gfCNCPoint5[18041] = {X 248.0563, Y 60.9282, Z -7.1667, A 0.000, B 0.000, C 0.000 }
gfCNCPoint5[18042] = {X 275.7918, Y 71.9370, Z -7.1667, A 0.000, B 0.000, C 0.000 }
gfCNCPoint5[18043] = {X 275.7935, Y 63.0708, Z -7.1667, A 0.000, B 0.000, C 0.000 }
gfCNCPoint5[18044] = {X 275.6909, Y 63.0586, Z -7.1667, A 0.000, B 0.000, C 0.000 }
gfCNCPoint5[18045] = {X 275.5887, Y 63.0439, Z -7.1667, A 0.000, B 0.000, C 0.000 }
gfCNCPoint5[18046] = {X 274.6513, Y 62.7818, Z -7.1667, A 0.000, B 0.000, C 0.000 }
gfCNCPoint5[18047] = {X 273.8005, Y 62.3090, Z -7.1667, A 0.000, B 0.000, C 0.000 }
gfCNCPoint5[18048] = {X 273.0828, Y 61.6514, Z -7.1667, A 0.000, B 0.000, C 0.000 }
gfCNCPoint5[18049] = {X 272.5376, Y 60.8451, Z -7.1667, A 0.000, B 0.000, C 0.000 }
gfCNCPoint5[18050] = {X 272.1947, Y 59.9341, Z -7.1667, A 0.000, B 0.000, C 0.000 }
gfCNCPoint5[18051] = {X 272.0728, Y 58.9684, Z -7.1667, A 0.000, B 0.000, C 0.000 }
gfCNCPoint5[18052] = {X 272.0727, Y 58.0000, Z -7.1667, A 0.000, B 0.000, C 0.000 }
gfCNCPoint5[18053] = {X 272.1770, Y 57.0743, Z -7.1667, A 0.000, B 0.000, C 0.000 }
gfCNCPoint5[18054] = {X 272.4847, Y 56.1950, Z -7.1667, A 0.000, B 0.000, C 0.000 }
gfCNCPoint5[18055] = {X 272.9803, Y 55.4063, Z -7.1667, A 0.000, B 0.000, C 0.000 }
gfCNCPoint5[18056] = {X 273.6390, Y 54.7476, Z -7.1667, A 0.000, B 0.000, C 0.000 }
gfCNCPoint5[18057] = {X 274.4277, Y 54.2520, Z -7.1667, A 0.000, B 0.000, C 0.000 }
gfCNCPoint5[18058] = {X 275.3070, Y 53.9443, Z -7.1667, A 0.000, B 0.000, C 0.000 }
gfCNCPoint5[18059] = {X 276.2327, Y 53.8400, Z -7.1667, A 0.000, B 0.000, C 0.000 }
gfCNCPoint5[18060] = {X 292.7731, Y 53.8400, Z -7.1667, A 0.000, B 0.000, C 0.000 }
gfCNCPoint5[18061] = {X 293.6988, Y 53.9443, Z -7.1667, A 0.000, B 0.000, C 0.000 }
gfCNCPoint5[18062] = {X 294.5780, Y 54.2520, Z -7.1667, A 0.000, B 0.000, C 0.000 }
gfCNCPoint5[18063] = {X 295.3668, Y 54.7476, Z -7.1667, A 0.000, B 0.000, C 0.000 }
gfCNCPoint5[18064] = {X 296.0255, Y 55.4063, Z -7.1667, A 0.000, B 0.000, C 0.000 }
gfCNCPoint5[18065] = {X 296.5211, Y 56.1950, Z -7.1667, A 0.000, B 0.000, C 0.000 }
gfCNCPoint5[18066] = {X 296.8288, Y 57.0743, Z -7.1667, A 0.000, B 0.000, C 0.000 }
gfCNCPoint5[18067] = {X 296.9331, Y 58.0000, Z -7.1667, A 0.000, B 0.000, C 0.000 }
gfCNCPoint5[18068] = {X 296.9331, Y 58.9345, Z -7.1667, A 0.000, B 0.000, C 0.000 }
gfCNCPoint5[18069] = {X 296.8157, Y 59.9063, Z -7.1667, A 0.000, B 0.000, C 0.000 }
gfCNCPoint5[18070] = {X 296.4753, Y 60.8241, Z -7.1667, A 0.000, B 0.000, C 0.000 }
gfCNCPoint5[18071] = {X 295.9306, Y 61.6374, Z -7.1667, A 0.000, B 0.000, C 0.000 }
gfCNCPoint5[18072] = {X 295.2116, Y 62.3015, Z -7.1667, A 0.000, B 0.000, C 0.000 }
gfCNCPoint5[18073] = {X 294.3577, Y 62.7801, Z -7.1667, A 0.000, B 0.000, C 0.000 }
gfCNCPoint5[18074] = {X 293.4159, Y 63.0468, Z -7.1667, A 0.000, B 0.000, C 0.000 }
gfCNCPoint5[18075] = {X 293.3191, Y 63.0611, Z -7.1667, A 0.000, B 0.000, C 0.000 }
gfCNCPoint5[18076] = {X 293.2221, Y 63.0731, Z -7.1667, A 0.000, B 0.000, C 0.000 }
gfCNCPoint5[18077] = {X 293.2138, Y 63.1615, Z -7.1667, A 0.000, B 0.000, C 0.000 }
gfCNCPoint5[18078] = {X 293.2249, Y 92.9203, Z -7.1667, A 0.000, B 0.000, C 0.000 }
gfCNCPoint5[18079] = {X 293.3202, Y 92.9325, Z -7.1667, A 0.000, B 0.000, C 0.000 }
gfCNCPoint5[18080] = {X 293.4152, Y 92.9468, Z -7.1667, A 0.000, B 0.000, C 0.000 }
gfCNCPoint5[18081] = {X 294.3566, Y 93.2161, Z -7.1667, A 0.000, B 0.000, C 0.000 }
gfCNCPoint5[18082] = {X 295.2099, Y 93.6965, Z -7.1667, A 0.000, B 0.000, C 0.000 }
gfCNCPoint5[18083] = {X 295.9285, Y 94.3617, Z -7.1667, A 0.000, B 0.000, C 0.000 }
gfCNCPoint5[18084] = {X 296.4732, Y 95.1754, Z -7.1667, A 0.000, B 0.000, C 0.000 }
gfCNCPoint5[18085] = {X 296.8142, Y 96.0933, Z -7.1667, A 0.000, B 0.000, C 0.000 }
gfCNCPoint5[18086] = {X 296.9331, Y 97.0653, Z -7.1667, A 0.000, B 0.000, C 0.000 }
gfCNCPoint5[18087] = {X 296.9331, Y 98.0000, Z -7.1667, A 0.000, B 0.000, C 0.000 }
gfCNCPoint5[18088] = {X 296.8288, Y 98.9257, Z -7.1667, A 0.000, B 0.000, C 0.000 }
gfCNCPoint5[18089] = {X 296.5211, Y 99.8050, Z -7.1667, A 0.000, B 0.000, C 0.000 }
gfCNCPoint5[18090] = {X 296.0255, Y 100.5937, Z -7.1667, A 0.000, B 0.000, C 0.000 }
gfCNCPoint5[18091] = {X 295.3668, Y 101.2524, Z -7.1667, A 0.000, B 0.000, C 0.000 }
gfCNCPoint5[18092] = {X 294.5780, Y 101.7480, Z -7.1667, A 0.000, B 0.000, C 0.000 }
gfCNCPoint5[18093] = {X 293.6988, Y 102.0557, Z -7.1667, A 0.000, B 0.000, C 0.000 }
gfCNCPoint5[18094] = {X 292.7731, Y 102.1600, Z -7.1667, A 0.000, B 0.000, C 0.000 }
gfCNCPoint5[18095] = {X 276.2327, Y 102.1600, Z -7.1667, A 0.000, B 0.000, C 0.000 }
gfCNCPoint5[18096] = {X 275.3070, Y 102.0557, Z -7.1667, A 0.000, B 0.000, C 0.000 }
gfCNCPoint5[18097] = {X 274.4277, Y 101.7480, Z -7.1667, A 0.000, B 0.000, C 0.000 }
gfCNCPoint5[18098] = {X 273.6390, Y 101.2524, Z -7.1667, A 0.000, B 0.000, C 0.000 }
gfCNCPoint5[18099] = {X 272.9803, Y 100.5937, Z -7.1667, A 0.000, B 0.000, C 0.000 }
gfCNCPoint5[18100] = {X 272.4847, Y 99.8050, Z -7.1667, A 0.000, B 0.000, C 0.000 }
gfCNCPoint5[18101] = {X 272.1770, Y 98.9257, Z -7.1667, A 0.000, B 0.000, C 0.000 }
gfCNCPoint5[18102] = {X 272.0727, Y 98.0000, Z -7.1667, A 0.000, B 0.000, C 0.000 }
gfCNCPoint5[18103] = {X 272.0727, Y 97.0658, Z -7.1667, A 0.000, B 0.000, C 0.000 }
gfCNCPoint5[18104] = {X 272.1634, Y 96.2021, Z -7.1667, A 0.000, B 0.000, C 0.000 }
gfCNCPoint5[18105] = {X 272.4314, Y 95.3761, Z -7.1667, A 0.000, B 0.000, C 0.000 }
gfCNCPoint5[18106] = {X 272.8651, Y 94.6237, Z -7.1667, A 0.000, B 0.000, C 0.000 }
gfCNCPoint5[18107] = {X 273.4455, Y 93.9777, Z -7.1667, A 0.000, B 0.000, C 0.000 }
gfCNCPoint5[18108] = {X 274.1475, Y 93.4663, Z -7.1667, A 0.000, B 0.000, C 0.000 }
gfCNCPoint5[18109] = {X 274.9403, Y 93.1118, Z -7.1667, A 0.000, B 0.000, C 0.000 }
gfCNCPoint5[18110] = {X 275.7894, Y 92.9296, Z -7.1667, A 0.000, B 0.000, C 0.000 }
gfCNCPoint5[18111] = {X 275.7894, Y 85.4858, Z -7.1667, A 0.000, B 0.000, C 0.000 }
gfCNCPoint5[18112] = {X 262.6229, Y 80.3245, Z -7.1667, A 0.000, B 0.000, C 0.000 }
gfCNCPoint5[18113] = {X 262.1919, Y 80.5968, Z -7.1667, A 0.000, B 0.000, C 0.000 }
gfCNCPoint5[18114] = {X 237.6370, Y 96.5016, Z -7.1667, A 0.000, B 0.000, C 0.000 }
gfCNCPoint5[18115] = {X 237.6398, Y 97.0655, Z -7.1667, A 0.000, B 0.000, C 0.000 }
gfCNCPoint5[18116] = {X 237.6398, Y 98.0000, Z -7.1667, A 0.000, B 0.000, C 0.000 }
gfCNCPoint5[18117] = {X 237.5355, Y 98.9257, Z -7.1667, A 0.000, B 0.000, C 0.000 }
gfCNCPoint5[18118] = {X 237.2278, Y 99.8050, Z -7.1667, A 0.000, B 0.000, C 0.000 }
gfCNCPoint5[18119] = {X 236.7322, Y 100.5937, Z -7.1667, A 0.000, B 0.000, C 0.000 }
gfCNCPoint5[18120] = {X 236.0735, Y 101.2524, Z -7.1667, A 0.000, B 0.000, C 0.000 }
gfCNCPoint5[18121] = {X 235.2847, Y 101.7480, Z -7.1667, A 0.000, B 0.000, C 0.000 }
gfCNCPoint5[18122] = {X 234.4055, Y 102.0557, Z -7.1667, A 0.000, B 0.000, C 0.000 }
gfCNCPoint5[18123] = {X 233.4798, Y 102.1600, Z -7.1667, A 0.000, B 0.000, C 0.000 }
gfCNCPoint5[18124] = {X 214.1790, Y 102.1600, Z -7.1667, A 0.000, B 0.000, C 0.000 }
gfCNCPoint5[18125] = {X 213.7860, Y 102.1414, Z -7.1667, A 0.000, B 0.000, C 0.000 }
gfCNCPoint5[18126] = {X 213.3966, Y 102.0857, Z -7.1667, A 0.000, B 0.000, C 0.000 }
gfCNCPoint5[18127] = {X 213.0071, Y 102.1414, Z -7.1667, A 0.000, B 0.000, C 0.000 }
gfCNCPoint5[18128] = {X 212.6141, Y 102.1600, Z -7.1667, A 0.000, B 0.000, C 0.000 }
gfCNCPoint5[18129] = {X 194.9870, Y 102.1600, Z -7.1667, A 0.000, B 0.000, C 0.000 }
gfCNCPoint5[18130] = {X 194.0613, Y 102.0557, Z -7.1667, A 0.000, B 0.000, C 0.000 }
gfCNCPoint5[18131] = {X 193.1820, Y 101.7480, Z -7.1667, A 0.000, B 0.000, C 0.000 }
gfCNCPoint5[18132] = {X 192.3932, Y 101.2524, Z -7.1667, A 0.000, B 0.000, C 0.000 }
gfCNCPoint5[18133] = {X 191.7345, Y 100.5937, Z -7.1667, A 0.000, B 0.000, C 0.000 }
gfCNCPoint5[18134] = {X 191.2389, Y 99.8050, Z -7.1667, A 0.000, B 0.000, C 0.000 }
gfCNCPoint5[18135] = {X 190.9313, Y 98.9257, Z -7.1667, A 0.000, B 0.000, C 0.000 }
gfCNCPoint5[18136] = {X 190.8270, Y 98.0000, Z -7.1667, A 0.000, B 0.000, C 0.000 }
gfCNCPoint5[18137] = {X 190.8270, Y 97.0659, Z -7.1667, A 0.000, B 0.000, C 0.000 }
gfCNCPoint5[18138] = {X 190.9241, Y 96.1723, Z -7.1667, A 0.000, B 0.000, C 0.000 }
gfCNCPoint5[18139] = {X 191.2109, Y 95.3203, Z -7.1667, A 0.000, B 0.000, C 0.000 }
gfCNCPoint5[18140] = {X 191.6741, Y 94.5499, Z -7.1667, A 0.000, B 0.000, C 0.000 }
gfCNCPoint5[18141] = {X 191.7354, Y 94.4712, Z -7.1667, A 0.000, B 0.000, C 0.000 }
gfCNCPoint5[18142] = {X 191.7986, Y 94.3939, Z -7.1667, A 0.000, B 0.000, C 0.000 }
gfCNCPoint5[18143] = {X 188.6351, Y 90.9402, Z -7.1667, A 0.000, B 0.000, C 0.000 }
gfCNCPoint5[18144] = {X 150.0187, Y 90.9402, Z -7.1667, A 0.000, B 0.000, C 0.000 }
gfCNCPoint5[18145] = {X 146.9341, Y 94.3576, Z -7.1667, A 0.000, B 0.000, C 0.000 }
gfCNCPoint5[18146] = {X 147.4805, Y 95.1722, Z -7.1667, A 0.000, B 0.000, C 0.000 }
gfCNCPoint5[18147] = {X 147.8218, Y 96.0918, Z -7.1667, A 0.000, B 0.000, C 0.000 }
gfCNCPoint5[18148] = {X 147.9391, Y 97.0657, Z -7.1667, A 0.000, B 0.000, C 0.000 }
gfCNCPoint5[18149] = {X 147.9391, Y 98.0000, Z -7.1667, A 0.000, B 0.000, C 0.000 }
gfCNCPoint5[18150] = {X 147.8348, Y 98.9257, Z -7.1667, A 0.000, B 0.000, C 0.000 }
gfCNCPoint5[18151] = {X 147.5271, Y 99.8050, Z -7.1667, A 0.000, B 0.000, C 0.000 }
gfCNCPoint5[18152] = {X 147.0315, Y 100.5937, Z -7.1667, A 0.000, B 0.000, C 0.000 }
gfCNCPoint5[18153] = {X 146.3728, Y 101.2524, Z -7.1667, A 0.000, B 0.000, C 0.000 }
gfCNCPoint5[18154] = {X 145.5841, Y 101.7480, Z -7.1667, A 0.000, B 0.000, C 0.000 }
gfCNCPoint5[18155] = {X 144.7048, Y 102.0557, Z -7.1667, A 0.000, B 0.000, C 0.000 }
gfCNCPoint5[18156] = {X 143.7791, Y 102.1600, Z -7.1667, A 0.000, B 0.000, C 0.000 }
gfCNCPoint5[18157] = {X 125.0000, Y 102.1600, Z -7.1667, A 0.000, B 0.000, C 0.000 }
gfCNCPoint5[18158] = {X 124.0743, Y 102.0557, Z -7.1667, A 0.000, B 0.000, C 0.000 }
gfCNCPoint5[18159] = {X 123.1950, Y 101.7480, Z -7.1667, A 0.000, B 0.000, C 0.000 }
gfCNCPoint5[18160] = {X 122.4063, Y 101.2524, Z -7.1667, A 0.000, B 0.000, C 0.000 }
gfCNCPoint5[18161] = {X 121.7476, Y 100.5937, Z -7.1667, A 0.000, B 0.000, C 0.000 }
gfCNCPoint5[18162] = {X 121.2520, Y 99.8050, Z -7.1667, A 0.000, B 0.000, C 0.000 }
gfCNCPoint5[18163] = {X 120.9443, Y 98.9257, Z -7.1667, A 0.000, B 0.000, C 0.000 }
gfCNCPoint5[18164] = {X 120.8400, Y 98.0000, Z -7.1667, A 0.000, B 0.000, C 0.000 }
gfCNCPoint5[18165] = {X 120.8400, Y 97.0659, Z -7.1667, A 0.000, B 0.000, C 0.000 }
gfCNCPoint5[18166] = {X 120.9405, Y 96.1569, Z -7.1667, A 0.000, B 0.000, C 0.000 }
gfCNCPoint5[18167] = {X 121.2373, Y 95.2918, Z -7.1667, A 0.000, B 0.000, C 0.000 }
gfCNCPoint5[18168] = {X 121.7159, Y 94.5125, Z -7.1667, A 0.000, B 0.000, C 0.000 }
gfCNCPoint5[18169] = {X 122.3532, Y 93.8566, Z -7.1667, A 0.000, B 0.000, C 0.000 }
gfCNCPoint5[18170] = {X 123.1185, Y 93.3558, Z -7.1667, A 0.000, B 0.000, C 0.000 }
gfCNCPoint5[18171] = {X 123.9747, Y 93.0343, Z -7.1667, A 0.000, B 0.000, C 0.000 }
gfCNCPoint5[18172] = {X 124.8804, Y 92.9077, Z -7.1667, A 0.000, B 0.000, C 0.000 }
gfCNCPoint5[18173] = {X 124.9141, Y 92.8889, Z -7.1667, A 0.000, B 0.000, C 0.000 }
gfCNCPoint5[18174] = {X 124.9512, Y 92.8787, Z -7.1667, A 0.000, B 0.000, C 0.000 }
gfCNCPoint5[18175] = {X 125.4723, Y 92.8015, Z -7.1667, A 0.000, B 0.000, C 0.000 }
gfCNCPoint5[18176] = {X 126.3315, Y 92.6561, Z -7.1667, A 0.000, B 0.000, C 0.000 }
gfCNCPoint5[18177] = {X 127.1785, Y 92.4511, Z -7.1667, A 0.000, B 0.000, C 0.000 }
gfCNCPoint5[18178] = {X 128.3866, Y 91.3174, Z -7.1667, A 0.000, B 0.000, C 0.000 }
gfCNCPoint5[18179] = {X 129.5302, Y 90.1187, Z -7.1667, A 0.000, B 0.000, C 0.000 }
gfCNCPoint5[18180] = {X 140.7977, Y 77.7462, Z -7.1667, A 0.000, B 0.000, C 0.000 }
gfCNCPoint5[18181] = {X 137.8403, Y 75.0529, Z -7.1667, A 0.000, B 0.000, C 0.000 }
gfCNCPoint5[18182] = {X 140.8568, Y 77.8000, Z -7.1667, A 0.000, B 0.000, C 0.000 }
gfCNCPoint5[18183] = {X 155.9346, Y 61.2436, Z -7.1667, A 0.000, B 0.000, C 0.000 }
gfCNCPoint5[18184] = {X 155.5463, Y 60.5376, Z -7.1667, A 0.000, B 0.000, C 0.000 }
gfCNCPoint5[18185] = {X 155.3043, Y 59.7689, Z -7.1667, A 0.000, B 0.000, C 0.000 }
gfCNCPoint5[18186] = {X 155.2181, Y 58.9678, Z -7.1667, A 0.000, B 0.000, C 0.000 }
gfCNCPoint5[18187] = {X 155.2180, Y 58.0000, Z -7.1667, A 0.000, B 0.000, C 0.000 }
gfCNCPoint5[18188] = {X 155.3203, Y 57.0921, Z -7.1667, A 0.000, B 0.000, C 0.000 }
gfCNCPoint5[18189] = {X 155.6220, Y 56.2298, Z -7.1667, A 0.000, B 0.000, C 0.000 }
gfCNCPoint5[18190] = {X 156.1081, Y 55.4562, Z -7.1667, A 0.000, B 0.000, C 0.000 }
gfCNCPoint5[18191] = {X 156.7541, Y 54.8101, Z -7.1667, A 0.000, B 0.000, C 0.000 }
gfCNCPoint5[18192] = {X 157.5277, Y 54.3240, Z -7.1667, A 0.000, B 0.000, C 0.000 }
gfCNCPoint5[18193] = {X 158.3901, Y 54.0223, Z -7.1667, A 0.000, B 0.000, C 0.000 }
gfCNCPoint5[18194] = {X 159.2980, Y 53.9200, Z -7.1667, A 0.000, B 0.000, C 0.000 }
gfCNCPoint5[18195] = {X 178.5335, Y 53.9200, Z -7.1667, A 0.000, B 0.000, C 0.000 }
gfCNCPoint5[18196] = {X 179.4414, Y 54.0223, Z -7.1667, A 0.000, B 0.000, C 0.000 }
gfCNCPoint5[18197] = {X 180.3037, Y 54.3240, Z -7.1667, A 0.000, B 0.000, C 0.000 }
gfCNCPoint5[18198] = {X 181.0773, Y 54.8101, Z -7.1667, A 0.000, B 0.000, C 0.000 }
gfCNCPoint5[18199] = {X 181.7234, Y 55.4562, Z -7.1667, A 0.000, B 0.000, C 0.000 }
gfCNCPoint5[18200] = {X 182.2095, Y 56.2298, Z -7.1667, A 0.000, B 0.000, C 0.000 }
gfCNCPoint5[18201] = {X 182.5112, Y 57.0921, Z -7.1667, A 0.000, B 0.000, C 0.000 }
gfCNCPoint5[18202] = {X 182.6135, Y 58.0000, Z -7.1667, A 0.000, B 0.000, C 0.000 }
gfCNCPoint5[18203] = {X 182.6135, Y 58.9342, Z -7.1667, A 0.000, B 0.000, C 0.000 }
gfCNCPoint5[18204] = {X 182.5335, Y 59.7381, Z -7.1667, A 0.000, B 0.000, C 0.000 }
gfCNCPoint5[18205] = {X 182.2967, Y 60.5104, Z -7.1667, A 0.000, B 0.000, C 0.000 }
gfCNCPoint5[18206] = {X 181.9123, Y 61.2210, Z -7.1667, A 0.000, B 0.000, C 0.000 }
gfCNCPoint5[18207] = {X 209.1194, Y 90.9217, Z -7.1667, A 0.000, B 0.000, C 0.000 }
gfCNCPoint5[18208] = {X 209.7993, Y 91.6258, Z -7.1667, A 0.000, B 0.000, C 0.000 }
gfCNCPoint5[18209] = {X 210.5151, Y 92.2933, Z -7.1667, A 0.000, B 0.000, C 0.000 }
gfCNCPoint5[18210] = {X 210.9595, Y 92.5941, Z -7.1667, A 0.000, B 0.000, C 0.000 }
gfCNCPoint5[18211] = {X 211.4659, Y 92.7713, Z -7.1667, A 0.000, B 0.000, C 0.000 }
gfCNCPoint5[18212] = {X 212.0678, Y 92.8979, Z -7.1667, A 0.000, B 0.000, C 0.000 }
gfCNCPoint5[18213] = {X 213.3902, Y 93.0645, Z -7.1667, A 0.000, B 0.000, C 0.000 }
gfCNCPoint5[18214] = {X 213.4129, Y 93.0582, Z -7.1667, A 0.000, B 0.000, C 0.000 }
gfCNCPoint5[18215] = {X 214.4629, Y 92.9753, Z -7.1667, A 0.000, B 0.000, C 0.000 }
gfCNCPoint5[18216] = {X 215.5144, Y 92.9145, Z -7.1667, A 0.000, B 0.000, C 0.000 }
gfCNCPoint5[18217] = {X 216.2276, Y 92.8363, Z -7.1667, A 0.000, B 0.000, C 0.000 }
gfCNCPoint5[18218] = {X 216.9142, Y 92.6283, Z -7.1667, A 0.000, B 0.000, C 0.000 }
gfCNCPoint5[18219] = {X 217.5510, Y 92.2978, Z -7.1667, A 0.000, B 0.000, C 0.000 }
gfCNCPoint5[18220] = {X 223.0910, Y 88.7225, Z -7.1667, A 0.000, B 0.000, C 0.000 }
gfCNCPoint5[18221] = {X 246.3530, Y 73.8482, Z -7.1667, A 0.000, B 0.000, C 0.000 }
gfCNCPoint5[18222] = {X 221.7196, Y 64.1819, Z -7.1667, A 0.000, B 0.000, C 0.000 }
gfCNCPoint5[18223] = {X 219.9261, Y 63.5817, Z -7.1667, A 0.000, B 0.000, C 0.000 }
gfCNCPoint5[18224] = {X 218.0758, Y 63.1899, Z -7.1667, A 0.000, B 0.000, C 0.000 }
gfCNCPoint5[18225] = {X 216.1929, Y 63.0117, Z -7.1667, A 0.000, B 0.000, C 0.000 }
gfCNCPoint5[18226] = {X 215.3127, Y 62.8850, Z -7.1667, A 0.000, B 0.000, C 0.000 }
gfCNCPoint5[18227] = {X 214.4809, Y 62.5706, Z -7.1667, A 0.000, B 0.000, C 0.000 }
gfCNCPoint5[18228] = {X 213.7369, Y 62.0834, Z -7.1667, A 0.000, B 0.000, C 0.000 }
gfCNCPoint5[18229] = {X 213.1162, Y 61.4466, Z -7.1667, A 0.000, B 0.000, C 0.000 }
gfCNCPoint5[18230] = {X 212.6482, Y 60.6905, Z -7.1667, A 0.000, B 0.000, C 0.000 }
gfCNCPoint5[18231] = {X 212.3552, Y 59.8509, Z -7.1667, A 0.000, B 0.000, C 0.000 }
gfCNCPoint5[18232] = {X 212.2509, Y 58.9678, Z -7.1667, A 0.000, B 0.000, C 0.000 }
gfCNCPoint5[18233] = {X 212.2508, Y 58.0000, Z -7.1667, A 0.000, B 0.000, C 0.000 }
gfCNCPoint5[18234] = {X 212.3531, Y 57.0921, Z -7.1667, A 0.000, B 0.000, C 0.000 }
gfCNCPoint5[18235] = {X 212.6549, Y 56.2298, Z -7.1667, A 0.000, B 0.000, C 0.000 }
gfCNCPoint5[18236] = {X 213.1409, Y 55.4562, Z -7.1667, A 0.000, B 0.000, C 0.000 }
gfCNCPoint5[18237] = {X 213.7870, Y 54.8101, Z -7.1667, A 0.000, B 0.000, C 0.000 }
gfCNCPoint5[18238] = {X 214.5606, Y 54.3240, Z -7.1667, A 0.000, B 0.000, C 0.000 }
gfCNCPoint5[18239] = {X 215.4229, Y 54.0223, Z -7.1667, A 0.000, B 0.000, C 0.000 }
gfCNCPoint5[18240] = {X 216.3308, Y 53.9200, Z -7.1667, A 0.000, B 0.000, C 0.000 }
gfCNCPoint5[18241] = {X 237.2617, Y 53.9200, Z -7.1667, A 0.000, B 0.000, C 0.000 }
gfCNCPoint5[18242] = {X 238.1696, Y 54.0223, Z -7.1667, A 0.000, B 0.000, C 0.000 }
gfCNCPoint5[18243] = {X 239.0319, Y 54.3240, Z -7.1667, A 0.000, B 0.000, C 0.000 }
gfCNCPoint5[18244] = {X 239.8055, Y 54.8101, Z -7.1667, A 0.000, B 0.000, C 0.000 }
gfCNCPoint5[18245] = {X 240.4516, Y 55.4562, Z -7.1667, A 0.000, B 0.000, C 0.000 }
gfCNCPoint5[18246] = {X 240.9376, Y 56.2298, Z -7.1667, A 0.000, B 0.000, C 0.000 }
gfCNCPoint5[18247] = {X 241.2394, Y 57.0921, Z -7.1667, A 0.000, B 0.000, C 0.000 }
gfCNCPoint5[18248] = {X 241.3417, Y 58.0000, Z -7.1667, A 0.000, B 0.000, C 0.000 }
gfCNCPoint5[18249] = {X 241.3417, Y 58.3958, Z -7.1667, A 0.000, B 0.000, C 0.000 }
gfCNCPoint5[18250] = {X 248.0270, Y 61.0026, Z -7.1667, A 0.000, B 0.000, C 0.000 }
gfCNCPoint5[18251] = {X 275.8718, Y 72.0548, Z -7.1667, A 0.000, B 0.000, C 0.000 }
gfCNCPoint5[18252] = {X 275.8735, Y 62.9982, Z -7.1667, A 0.000, B 0.000, C 0.000 }
gfCNCPoint5[18253] = {X 275.7370, Y 62.9838, Z -7.1667, A 0.000, B 0.000, C 0.000 }
gfCNCPoint5[18254] = {X 275.6011, Y 62.9649, Z -7.1667, A 0.000, B 0.000, C 0.000 }
gfCNCPoint5[18255] = {X 274.6817, Y 62.7078, Z -7.1667, A 0.000, B 0.000, C 0.000 }
gfCNCPoint5[18256] = {X 273.8473, Y 62.2441, Z -7.1667, A 0.000, B 0.000, C 0.000 }
gfCNCPoint5[18257] = {X 273.1434, Y 61.5992, Z -7.1667, A 0.000, B 0.000, C 0.000 }
gfCNCPoint5[18258] = {X 272.6087, Y 60.8083, Z -7.1667, A 0.000, B 0.000, C 0.000 }
gfCNCPoint5[18259] = {X 272.2723, Y 59.9149, Z -7.1667, A 0.000, B 0.000, C 0.000 }
gfCNCPoint5[18260] = {X 272.1528, Y 58.9678, Z -7.1667, A 0.000, B 0.000, C 0.000 }
gfCNCPoint5[18261] = {X 272.1527, Y 58.0000, Z -7.1667, A 0.000, B 0.000, C 0.000 }
gfCNCPoint5[18262] = {X 272.2550, Y 57.0921, Z -7.1667, A 0.000, B 0.000, C 0.000 }
gfCNCPoint5[18263] = {X 272.5567, Y 56.2298, Z -7.1667, A 0.000, B 0.000, C 0.000 }
gfCNCPoint5[18264] = {X 273.0428, Y 55.4562, Z -7.1667, A 0.000, B 0.000, C 0.000 }
gfCNCPoint5[18265] = {X 273.6889, Y 54.8101, Z -7.1667, A 0.000, B 0.000, C 0.000 }
gfCNCPoint5[18266] = {X 274.4624, Y 54.3240, Z -7.1667, A 0.000, B 0.000, C 0.000 }
gfCNCPoint5[18267] = {X 275.3248, Y 54.0223, Z -7.1667, A 0.000, B 0.000, C 0.000 }
gfCNCPoint5[18268] = {X 276.2327, Y 53.9200, Z -7.1667, A 0.000, B 0.000, C 0.000 }
gfCNCPoint5[18269] = {X 292.7731, Y 53.9200, Z -7.1667, A 0.000, B 0.000, C 0.000 }
gfCNCPoint5[18270] = {X 293.6810, Y 54.0223, Z -7.1667, A 0.000, B 0.000, C 0.000 }
gfCNCPoint5[18271] = {X 294.5433, Y 54.3240, Z -7.1667, A 0.000, B 0.000, C 0.000 }
gfCNCPoint5[18272] = {X 295.3169, Y 54.8101, Z -7.1667, A 0.000, B 0.000, C 0.000 }
gfCNCPoint5[18273] = {X 295.9630, Y 55.4562, Z -7.1667, A 0.000, B 0.000, C 0.000 }
gfCNCPoint5[18274] = {X 296.4490, Y 56.2298, Z -7.1667, A 0.000, B 0.000, C 0.000 }
gfCNCPoint5[18275] = {X 296.7508, Y 57.0921, Z -7.1667, A 0.000, B 0.000, C 0.000 }
gfCNCPoint5[18276] = {X 296.8531, Y 58.0000, Z -7.1667, A 0.000, B 0.000, C 0.000 }
gfCNCPoint5[18277] = {X 296.8531, Y 58.9343, Z -7.1667, A 0.000, B 0.000, C 0.000 }
gfCNCPoint5[18278] = {X 296.7379, Y 59.8875, Z -7.1667, A 0.000, B 0.000, C 0.000 }
gfCNCPoint5[18279] = {X 296.4041, Y 60.7876, Z -7.1667, A 0.000, B 0.000, C 0.000 }
gfCNCPoint5[18280] = {X 295.8698, Y 61.5854, Z -7.1667, A 0.000, B 0.000, C 0.000 }
gfCNCPoint5[18281] = {X 295.1646, Y 62.2368, Z -7.1667, A 0.000, B 0.000, C 0.000 }
gfCNCPoint5[18282] = {X 294.3271, Y 62.7062, Z -7.1667, A 0.000, B 0.000, C 0.000 }
gfCNCPoint5[18283] = {X 293.4033, Y 62.9678, Z -7.1667, A 0.000, B 0.000, C 0.000 }
gfCNCPoint5[18284] = {X 293.2762, Y 62.9860, Z -7.1667, A 0.000, B 0.000, C 0.000 }
gfCNCPoint5[18285] = {X 293.1486, Y 63.0003, Z -7.1667, A 0.000, B 0.000, C 0.000 }
gfCNCPoint5[18286] = {X 293.1338, Y 63.1578, Z -7.1667, A 0.000, B 0.000, C 0.000 }
gfCNCPoint5[18287] = {X 293.1449, Y 92.9921, Z -7.1667, A 0.000, B 0.000, C 0.000 }
gfCNCPoint5[18288] = {X 293.2739, Y 93.0069, Z -7.1667, A 0.000, B 0.000, C 0.000 }
gfCNCPoint5[18289] = {X 293.4023, Y 93.0258, Z -7.1667, A 0.000, B 0.000, C 0.000 }
gfCNCPoint5[18290] = {X 294.3258, Y 93.2900, Z -7.1667, A 0.000, B 0.000, C 0.000 }
gfCNCPoint5[18291] = {X 295.1628, Y 93.7612, Z -7.1667, A 0.000, B 0.000, C 0.000 }
gfCNCPoint5[18292] = {X 295.8677, Y 94.4136, Z -7.1667, A 0.000, B 0.000, C 0.000 }
gfCNCPoint5[18293] = {X 296.4019, Y 95.2119, Z -7.1667, A 0.000, B 0.000, C 0.000 }
gfCNCPoint5[18294] = {X 296.7365, Y 96.1122, Z -7.1667, A 0.000, B 0.000, C 0.000 }
gfCNCPoint5[18295] = {X 296.8531, Y 97.0657, Z -7.1667, A 0.000, B 0.000, C 0.000 }
gfCNCPoint5[18296] = {X 296.8531, Y 98.0000, Z -7.1667, A 0.000, B 0.000, C 0.000 }
gfCNCPoint5[18297] = {X 296.7508, Y 98.9079, Z -7.1667, A 0.000, B 0.000, C 0.000 }
gfCNCPoint5[18298] = {X 296.4490, Y 99.7702, Z -7.1667, A 0.000, B 0.000, C 0.000 }
gfCNCPoint5[18299] = {X 295.9630, Y 100.5438, Z -7.1667, A 0.000, B 0.000, C 0.000 }
gfCNCPoint5[18300] = {X 295.3169, Y 101.1899, Z -7.1667, A 0.000, B 0.000, C 0.000 }
gfCNCPoint5[18301] = {X 294.5433, Y 101.6760, Z -7.1667, A 0.000, B 0.000, C 0.000 }
gfCNCPoint5[18302] = {X 293.6810, Y 101.9777, Z -7.1667, A 0.000, B 0.000, C 0.000 }
gfCNCPoint5[18303] = {X 292.7731, Y 102.0800, Z -7.1667, A 0.000, B 0.000, C 0.000 }
gfCNCPoint5[18304] = {X 276.2327, Y 102.0800, Z -7.1667, A 0.000, B 0.000, C 0.000 }
gfCNCPoint5[18305] = {X 275.3248, Y 101.9777, Z -7.1667, A 0.000, B 0.000, C 0.000 }
gfCNCPoint5[18306] = {X 274.4624, Y 101.6760, Z -7.1667, A 0.000, B 0.000, C 0.000 }
gfCNCPoint5[18307] = {X 273.6889, Y 101.1899, Z -7.1667, A 0.000, B 0.000, C 0.000 }
gfCNCPoint5[18308] = {X 273.0428, Y 100.5438, Z -7.1667, A 0.000, B 0.000, C 0.000 }
gfCNCPoint5[18309] = {X 272.5567, Y 99.7702, Z -7.1667, A 0.000, B 0.000, C 0.000 }
gfCNCPoint5[18310] = {X 272.2550, Y 98.9079, Z -7.1667, A 0.000, B 0.000, C 0.000 }
gfCNCPoint5[18311] = {X 272.1527, Y 98.0000, Z -7.1667, A 0.000, B 0.000, C 0.000 }
gfCNCPoint5[18312] = {X 272.1527, Y 97.0658, Z -7.1667, A 0.000, B 0.000, C 0.000 }
gfCNCPoint5[18313] = {X 272.2438, Y 96.2087, Z -7.1667, A 0.000, B 0.000, C 0.000 }
gfCNCPoint5[18314] = {X 272.5129, Y 95.3898, Z -7.1667, A 0.000, B 0.000, C 0.000 }
gfCNCPoint5[18315] = {X 272.9480, Y 94.6458, Z -7.1667, A 0.000, B 0.000, C 0.000 }
gfCNCPoint5[18316] = {X 273.5297, Y 94.0097, Z -7.1667, A 0.000, B 0.000, C 0.000 }
gfCNCPoint5[18317] = {X 274.2321, Y 93.5101, Z -7.1667, A 0.000, B 0.000, C 0.000 }
gfCNCPoint5[18318] = {X 275.0238, Y 93.1692, Z -7.1667, A 0.000, B 0.000, C 0.000 }
gfCNCPoint5[18319] = {X 275.8694, Y 93.0021, Z -7.1667, A 0.000, B 0.000, C 0.000 }
gfCNCPoint5[18320] = {X 275.8694, Y 85.4313, Z -7.1667, A 0.000, B 0.000, C 0.000 }
gfCNCPoint5[18321] = {X 262.6144, Y 80.2353, Z -7.1667, A 0.000, B 0.000, C 0.000 }
gfCNCPoint5[18322] = {X 262.1488, Y 80.5294, Z -7.1667, A 0.000, B 0.000, C 0.000 }
gfCNCPoint5[18323] = {X 237.5567, Y 96.4583, Z -7.1667, A 0.000, B 0.000, C 0.000 }
gfCNCPoint5[18324] = {X 237.5598, Y 97.0657, Z -7.1667, A 0.000, B 0.000, C 0.000 }
gfCNCPoint5[18325] = {X 237.5598, Y 98.0000, Z -7.1667, A 0.000, B 0.000, C 0.000 }
gfCNCPoint5[18326] = {X 237.4575, Y 98.9079, Z -7.1667, A 0.000, B 0.000, C 0.000 }
gfCNCPoint5[18327] = {X 237.1557, Y 99.7702, Z -7.1667, A 0.000, B 0.000, C 0.000 }
gfCNCPoint5[18328] = {X 236.6697, Y 100.5438, Z -7.1667, A 0.000, B 0.000, C 0.000 }
gfCNCPoint5[18329] = {X 236.0236, Y 101.1899, Z -7.1667, A 0.000, B 0.000, C 0.000 }
gfCNCPoint5[18330] = {X 235.2500, Y 101.6760, Z -7.1667, A 0.000, B 0.000, C 0.000 }
gfCNCPoint5[18331] = {X 234.3877, Y 101.9777, Z -7.1667, A 0.000, B 0.000, C 0.000 }
gfCNCPoint5[18332] = {X 233.4798, Y 102.0800, Z -7.1667, A 0.000, B 0.000, C 0.000 }
gfCNCPoint5[18333] = {X 214.1790, Y 102.0800, Z -7.1667, A 0.000, B 0.000, C 0.000 }
gfCNCPoint5[18334] = {X 213.7860, Y 102.0610, Z -7.1667, A 0.000, B 0.000, C 0.000 }
gfCNCPoint5[18335] = {X 213.3966, Y 102.0043, Z -7.1667, A 0.000, B 0.000, C 0.000 }
gfCNCPoint5[18336] = {X 213.0072, Y 102.0610, Z -7.1667, A 0.000, B 0.000, C 0.000 }
gfCNCPoint5[18337] = {X 212.6141, Y 102.0800, Z -7.1667, A 0.000, B 0.000, C 0.000 }
gfCNCPoint5[18338] = {X 194.9870, Y 102.0800, Z -7.1667, A 0.000, B 0.000, C 0.000 }
gfCNCPoint5[18339] = {X 194.0791, Y 101.9777, Z -7.1667, A 0.000, B 0.000, C 0.000 }
gfCNCPoint5[18340] = {X 193.2167, Y 101.6760, Z -7.1667, A 0.000, B 0.000, C 0.000 }
gfCNCPoint5[18341] = {X 192.4431, Y 101.1899, Z -7.1667, A 0.000, B 0.000, C 0.000 }
gfCNCPoint5[18342] = {X 191.7971, Y 100.5438, Z -7.1667, A 0.000, B 0.000, C 0.000 }
gfCNCPoint5[18343] = {X 191.3110, Y 99.7702, Z -7.1667, A 0.000, B 0.000, C 0.000 }
gfCNCPoint5[18344] = {X 191.0093, Y 98.9079, Z -7.1667, A 0.000, B 0.000, C 0.000 }
gfCNCPoint5[18345] = {X 190.9070, Y 98.0000, Z -7.1667, A 0.000, B 0.000, C 0.000 }
gfCNCPoint5[18346] = {X 190.9070, Y 97.0659, Z -7.1667, A 0.000, B 0.000, C 0.000 }
gfCNCPoint5[18347] = {X 191.0022, Y 96.1894, Z -7.1667, A 0.000, B 0.000, C 0.000 }
gfCNCPoint5[18348] = {X 191.2835, Y 95.3539, Z -7.1667, A 0.000, B 0.000, C 0.000 }
gfCNCPoint5[18349] = {X 191.7378, Y 94.5983, Z -7.1667, A 0.000, B 0.000, C 0.000 }
gfCNCPoint5[18350] = {X 191.8199, Y 94.4938, Z -7.1667, A 0.000, B 0.000, C 0.000 }
gfCNCPoint5[18351] = {X 191.9053, Y 94.3920, Z -7.1667, A 0.000, B 0.000, C 0.000 }
gfCNCPoint5[18352] = {X 188.6703, Y 90.8602, Z -7.1667, A 0.000, B 0.000, C 0.000 }
gfCNCPoint5[18353] = {X 149.9831, Y 90.8602, Z -7.1667, A 0.000, B 0.000, C 0.000 }
gfCNCPoint5[18354] = {X 146.8272, Y 94.3567, Z -7.1667, A 0.000, B 0.000, C 0.000 }
gfCNCPoint5[18355] = {X 147.3877, Y 95.1671, Z -7.1667, A 0.000, B 0.000, C 0.000 }
gfCNCPoint5[18356] = {X 147.7384, Y 96.0879, Z -7.1667, A 0.000, B 0.000, C 0.000 }
gfCNCPoint5[18357] = {X 147.8591, Y 97.0659, Z -7.1667, A 0.000, B 0.000, C 0.000 }
gfCNCPoint5[18358] = {X 147.8591, Y 98.0000, Z -7.1667, A 0.000, B 0.000, C 0.000 }
gfCNCPoint5[18359] = {X 147.7568, Y 98.9079, Z -7.1667, A 0.000, B 0.000, C 0.000 }
gfCNCPoint5[18360] = {X 147.4551, Y 99.7702, Z -7.1667, A 0.000, B 0.000, C 0.000 }
gfCNCPoint5[18361] = {X 146.9690, Y 100.5438, Z -7.1667, A 0.000, B 0.000, C 0.000 }
gfCNCPoint5[18362] = {X 146.3229, Y 101.1899, Z -7.1667, A 0.000, B 0.000, C 0.000 }
gfCNCPoint5[18363] = {X 145.5494, Y 101.6760, Z -7.1667, A 0.000, B 0.000, C 0.000 }
gfCNCPoint5[18364] = {X 144.6870, Y 101.9777, Z -7.1667, A 0.000, B 0.000, C 0.000 }
gfCNCPoint5[18365] = {X 143.7791, Y 102.0800, Z -7.1667, A 0.000, B 0.000, C 0.000 }
gfCNCPoint5[18366] = {X 125.0000, Y 102.0800, Z -7.1667, A 0.000, B 0.000, C 0.000 }
gfCNCPoint5[18367] = {X 124.0921, Y 101.9777, Z -7.1667, A 0.000, B 0.000, C 0.000 }
gfCNCPoint5[18368] = {X 123.2298, Y 101.6760, Z -7.1667, A 0.000, B 0.000, C 0.000 }
gfCNCPoint5[18369] = {X 122.4562, Y 101.1899, Z -7.1667, A 0.000, B 0.000, C 0.000 }
gfCNCPoint5[18370] = {X 121.8101, Y 100.5438, Z -7.1667, A 0.000, B 0.000, C 0.000 }
gfCNCPoint5[18371] = {X 121.3240, Y 99.7702, Z -7.1667, A 0.000, B 0.000, C 0.000 }
gfCNCPoint5[18372] = {X 121.0223, Y 98.9079, Z -7.1667, A 0.000, B 0.000, C 0.000 }
gfCNCPoint5[18373] = {X 120.9200, Y 98.0000, Z -7.1667, A 0.000, B 0.000, C 0.000 }
gfCNCPoint5[18374] = {X 120.9200, Y 97.0659, Z -7.1667, A 0.000, B 0.000, C 0.000 }
gfCNCPoint5[18375] = {X 121.0193, Y 96.1711, Z -7.1667, A 0.000, B 0.000, C 0.000 }
gfCNCPoint5[18376] = {X 121.3125, Y 95.3198, Z -7.1667, A 0.000, B 0.000, C 0.000 }
gfCNCPoint5[18377] = {X 121.7853, Y 94.5536, Z -7.1667, A 0.000, B 0.000, C 0.000 }
gfCNCPoint5[18378] = {X 122.4145, Y 93.9097, Z -7.1667, A 0.000, B 0.000, C 0.000 }
gfCNCPoint5[18379] = {X 123.1697, Y 93.4195, Z -7.1667, A 0.000, B 0.000, C 0.000 }
gfCNCPoint5[18380] = {X 124.0140, Y 93.1069, Z -7.1667, A 0.000, B 0.000, C 0.000 }
gfCNCPoint5[18381] = {X 124.9064, Y 92.9870, Z -7.1667, A 0.000, B 0.000, C 0.000 }
gfCNCPoint5[18382] = {X 124.9291, Y 92.9713, Z -7.1667, A 0.000, B 0.000, C 0.000 }
gfCNCPoint5[18383] = {X 124.9629, Y 92.9579, Z -7.1667, A 0.000, B 0.000, C 0.000 }
gfCNCPoint5[18384] = {X 125.4829, Y 92.8808, Z -7.1667, A 0.000, B 0.000, C 0.000 }
gfCNCPoint5[18385] = {X 126.3567, Y 92.7327, Z -7.1667, A 0.000, B 0.000, C 0.000 }
gfCNCPoint5[18386] = {X 127.2178, Y 92.5232, Z -7.1667, A 0.000, B 0.000, C 0.000 }
gfCNCPoint5[18387] = {X 128.4364, Y 91.3807, Z -7.1667, A 0.000, B 0.000, C 0.000 }
gfCNCPoint5[18388] = {X 129.5896, Y 90.1723, Z -7.1667, A 0.000, B 0.000, C 0.000 }
gfCNCPoint5[18389] = {X 140.8568, Y 77.8000, Z -7.1667, A 0.000, B 0.000, C 0.000 }
gfCNCPoint5[18390] = {X 137.8994, Y 75.1068, Z -7.1667, A 0.000, B 0.000, C 0.000 }
gfCNCPoint5[18391] = {X 140.9160, Y 77.8539, Z -7.1667, A 0.000, B 0.000, C 0.000 }
gfCNCPoint5[18392] = {X 156.0368, Y 61.2502, Z -7.1667, A 0.000, B 0.000, C 0.000 }
gfCNCPoint5[18393] = {X 155.6322, Y 60.5347, Z -7.1667, A 0.000, B 0.000, C 0.000 }
gfCNCPoint5[18394] = {X 155.3824, Y 59.7517, Z -7.1667, A 0.000, B 0.000, C 0.000 }
gfCNCPoint5[18395] = {X 155.2980, Y 58.9341, Z -7.1667, A 0.000, B 0.000, C 0.000 }
gfCNCPoint5[18396] = {X 155.2980, Y 58.0000, Z -7.1667, A 0.000, B 0.000, C 0.000 }
gfCNCPoint5[18397] = {X 155.3982, Y 57.1099, Z -7.1667, A 0.000, B 0.000, C 0.000 }
gfCNCPoint5[18398] = {X 155.6941, Y 56.2645, Z -7.1667, A 0.000, B 0.000, C 0.000 }
gfCNCPoint5[18399] = {X 156.1706, Y 55.5060, Z -7.1667, A 0.000, B 0.000, C 0.000 }
gfCNCPoint5[18400] = {X 156.8040, Y 54.8727, Z -7.1667, A 0.000, B 0.000, C 0.000 }
gfCNCPoint5[18401] = {X 157.5624, Y 54.3961, Z -7.1667, A 0.000, B 0.000, C 0.000 }
gfCNCPoint5[18402] = {X 158.4079, Y 54.1003, Z -7.1667, A 0.000, B 0.000, C 0.000 }
gfCNCPoint5[18403] = {X 159.2980, Y 54.0000, Z -7.1667, A 0.000, B 0.000, C 0.000 }
gfCNCPoint5[18404] = {X 178.5335, Y 54.0000, Z -7.1667, A 0.000, B 0.000, C 0.000 }
gfCNCPoint5[18405] = {X 179.4236, Y 54.1003, Z -7.1667, A 0.000, B 0.000, C 0.000 }
gfCNCPoint5[18406] = {X 180.2690, Y 54.3961, Z -7.1667, A 0.000, B 0.000, C 0.000 }
gfCNCPoint5[18407] = {X 181.0275, Y 54.8727, Z -7.1667, A 0.000, B 0.000, C 0.000 }
gfCNCPoint5[18408] = {X 181.6608, Y 55.5060, Z -7.1667, A 0.000, B 0.000, C 0.000 }
gfCNCPoint5[18409] = {X 182.1374, Y 56.2645, Z -7.1667, A 0.000, B 0.000, C 0.000 }
gfCNCPoint5[18410] = {X 182.4332, Y 57.1099, Z -7.1667, A 0.000, B 0.000, C 0.000 }
gfCNCPoint5[18411] = {X 182.5335, Y 58.0000, Z -7.1667, A 0.000, B 0.000, C 0.000 }
gfCNCPoint5[18412] = {X 182.5334, Y 58.9671, Z -7.1667, A 0.000, B 0.000, C 0.000 }
gfCNCPoint5[18413] = {X 182.4464, Y 59.7644, Z -7.1667, A 0.000, B 0.000, C 0.000 }
gfCNCPoint5[18414] = {X 182.2021, Y 60.5283, Z -7.1667, A 0.000, B 0.000, C 0.000 }
gfCNCPoint5[18415] = {X 181.8103, Y 61.2281, Z -7.1667, A 0.000, B 0.000, C 0.000 }
gfCNCPoint5[18416] = {X 209.0604, Y 90.9758, Z -7.1667, A 0.000, B 0.000, C 0.000 }
gfCNCPoint5[18417] = {X 209.7432, Y 91.6829, Z -7.1667, A 0.000, B 0.000, C 0.000 }
gfCNCPoint5[18418] = {X 210.4621, Y 92.3532, Z -7.1667, A 0.000, B 0.000, C 0.000 }
gfCNCPoint5[18419] = {X 210.9235, Y 92.6655, Z -7.1667, A 0.000, B 0.000, C 0.000 }
gfCNCPoint5[18420] = {X 211.4495, Y 92.8496, Z -7.1667, A 0.000, B 0.000, C 0.000 }
gfCNCPoint5[18421] = {X 212.0545, Y 92.9769, Z -7.1667, A 0.000, B 0.000, C 0.000 }
gfCNCPoint5[18422] = {X 213.3962, Y 93.1459, Z -7.1667, A 0.000, B 0.000, C 0.000 }
gfCNCPoint5[18423] = {X 213.4273, Y 93.1372, Z -7.1667, A 0.000, B 0.000, C 0.000 }
gfCNCPoint5[18424] = {X 214.4714, Y 93.0549, Z -7.1667, A 0.000, B 0.000, C 0.000 }
gfCNCPoint5[18425] = {X 215.5170, Y 92.9945, Z -7.1667, A 0.000, B 0.000, C 0.000 }
gfCNCPoint5[18426] = {X 216.2444, Y 92.9145, Z -7.1667, A 0.000, B 0.000, C 0.000 }
gfCNCPoint5[18427] = {X 216.9449, Y 92.7023, Z -7.1667, A 0.000, B 0.000, C 0.000 }
gfCNCPoint5[18428] = {X 217.5944, Y 92.3650, Z -7.1667, A 0.000, B 0.000, C 0.000 }
gfCNCPoint5[18429] = {X 223.1343, Y 88.7898, Z -7.1667, A 0.000, B 0.000, C 0.000 }
gfCNCPoint5[18430] = {X 246.5283, Y 73.8311, Z -7.1667, A 0.000, B 0.000, C 0.000 }
gfCNCPoint5[18431] = {X 221.7493, Y 64.1076, Z -7.1667, A 0.000, B 0.000, C 0.000 }
gfCNCPoint5[18432] = {X 219.9471, Y 63.5045, Z -7.1667, A 0.000, B 0.000, C 0.000 }
gfCNCPoint5[18433] = {X 218.0878, Y 63.1108, Z -7.1667, A 0.000, B 0.000, C 0.000 }
gfCNCPoint5[18434] = {X 216.1958, Y 62.9318, Z -7.1667, A 0.000, B 0.000, C 0.000 }
gfCNCPoint5[18435] = {X 215.3283, Y 62.8064, Z -7.1667, A 0.000, B 0.000, C 0.000 }
gfCNCPoint5[18436] = {X 214.5089, Y 62.4951, Z -7.1667, A 0.000, B 0.000, C 0.000 }
gfCNCPoint5[18437] = {X 213.7770, Y 62.0127, Z -7.1667, A 0.000, B 0.000, C 0.000 }
gfCNCPoint5[18438] = {X 213.1677, Y 61.3825, Z -7.1667, A 0.000, B 0.000, C 0.000 }
gfCNCPoint5[18439] = {X 212.7104, Y 60.6348, Z -7.1667, A 0.000, B 0.000, C 0.000 }
gfCNCPoint5[18440] = {X 212.4268, Y 59.8053, Z -7.1667, A 0.000, B 0.000, C 0.000 }
gfCNCPoint5[18441] = {X 212.3308, Y 58.9341, Z -7.1667, A 0.000, B 0.000, C 0.000 }
gfCNCPoint5[18442] = {X 212.3308, Y 58.0000, Z -7.1667, A 0.000, B 0.000, C 0.000 }
gfCNCPoint5[18443] = {X 212.4311, Y 57.1099, Z -7.1667, A 0.000, B 0.000, C 0.000 }
gfCNCPoint5[18444] = {X 212.7269, Y 56.2645, Z -7.1667, A 0.000, B 0.000, C 0.000 }
gfCNCPoint5[18445] = {X 213.2035, Y 55.5060, Z -7.1667, A 0.000, B 0.000, C 0.000 }
gfCNCPoint5[18446] = {X 213.8368, Y 54.8727, Z -7.1667, A 0.000, B 0.000, C 0.000 }
gfCNCPoint5[18447] = {X 214.5953, Y 54.3961, Z -7.1667, A 0.000, B 0.000, C 0.000 }
gfCNCPoint5[18448] = {X 215.4407, Y 54.1003, Z -7.1667, A 0.000, B 0.000, C 0.000 }
gfCNCPoint5[18449] = {X 216.3308, Y 54.0000, Z -7.1667, A 0.000, B 0.000, C 0.000 }
gfCNCPoint5[18450] = {X 237.2617, Y 54.0000, Z -7.1667, A 0.000, B 0.000, C 0.000 }
gfCNCPoint5[18451] = {X 238.1518, Y 54.1003, Z -7.1667, A 0.000, B 0.000, C 0.000 }
gfCNCPoint5[18452] = {X 238.9972, Y 54.3961, Z -7.1667, A 0.000, B 0.000, C 0.000 }
gfCNCPoint5[18453] = {X 239.7556, Y 54.8727, Z -7.1667, A 0.000, B 0.000, C 0.000 }
gfCNCPoint5[18454] = {X 240.3890, Y 55.5060, Z -7.1667, A 0.000, B 0.000, C 0.000 }
gfCNCPoint5[18455] = {X 240.8656, Y 56.2645, Z -7.1667, A 0.000, B 0.000, C 0.000 }
gfCNCPoint5[18456] = {X 241.1614, Y 57.1099, Z -7.1667, A 0.000, B 0.000, C 0.000 }
gfCNCPoint5[18457] = {X 241.2617, Y 58.0000, Z -7.1667, A 0.000, B 0.000, C 0.000 }
gfCNCPoint5[18458] = {X 241.2617, Y 58.4504, Z -7.1667, A 0.000, B 0.000, C 0.000 }
gfCNCPoint5[18459] = {X 247.9977, Y 61.0771, Z -7.1667, A 0.000, B 0.000, C 0.000 }
gfCNCPoint5[18460] = {X 275.9518, Y 72.1726, Z -7.1667, A 0.000, B 0.000, C 0.000 }
gfCNCPoint5[18461] = {X 275.9515, Y 63.0394, Z -7.1667, A 0.000, B 0.000, C 0.000 }
gfCNCPoint5[18462] = {X 275.9573, Y 62.9246, Z -7.1667, A 0.000, B 0.000, C 0.000 }
gfCNCPoint5[18463] = {X 275.7850, Y 62.9089, Z -7.1667, A 0.000, B 0.000, C 0.000 }
gfCNCPoint5[18464] = {X 275.6135, Y 62.8858, Z -7.1667, A 0.000, B 0.000, C 0.000 }
gfCNCPoint5[18465] = {X 274.7070, Y 62.6317, Z -7.1667, A 0.000, B 0.000, C 0.000 }
gfCNCPoint5[18466] = {X 273.8851, Y 62.1727, Z -7.1667, A 0.000, B 0.000, C 0.000 }
gfCNCPoint5[18467] = {X 273.1932, Y 61.5344, Z -7.1667, A 0.000, B 0.000, C 0.000 }
gfCNCPoint5[18468] = {X 272.6697, Y 60.7520, Z -7.1667, A 0.000, B 0.000, C 0.000 }
gfCNCPoint5[18469] = {X 272.3435, Y 59.8689, Z -7.1667, A 0.000, B 0.000, C 0.000 }
gfCNCPoint5[18470] = {X 272.2327, Y 58.9341, Z -7.1667, A 0.000, B 0.000, C 0.000 }
gfCNCPoint5[18471] = {X 272.2327, Y 58.0000, Z -7.1667, A 0.000, B 0.000, C 0.000 }
gfCNCPoint5[18472] = {X 272.3330, Y 57.1099, Z -7.1667, A 0.000, B 0.000, C 0.000 }
gfCNCPoint5[18473] = {X 272.6288, Y 56.2645, Z -7.1667, A 0.000, B 0.000, C 0.000 }
gfCNCPoint5[18474] = {X 273.1054, Y 55.5060, Z -7.1667, A 0.000, B 0.000, C 0.000 }
gfCNCPoint5[18475] = {X 273.7387, Y 54.8727, Z -7.1667, A 0.000, B 0.000, C 0.000 }
gfCNCPoint5[18476] = {X 274.4972, Y 54.3961, Z -7.1667, A 0.000, B 0.000, C 0.000 }
gfCNCPoint5[18477] = {X 275.3426, Y 54.1003, Z -7.1667, A 0.000, B 0.000, C 0.000 }
gfCNCPoint5[18478] = {X 276.2327, Y 54.0000, Z -7.1667, A 0.000, B 0.000, C 0.000 }
gfCNCPoint5[18479] = {X 292.7731, Y 54.0000, Z -7.1667, A 0.000, B 0.000, C 0.000 }
gfCNCPoint5[18480] = {X 293.6632, Y 54.1003, Z -7.1667, A 0.000, B 0.000, C 0.000 }
gfCNCPoint5[18481] = {X 294.5086, Y 54.3961, Z -7.1667, A 0.000, B 0.000, C 0.000 }
gfCNCPoint5[18482] = {X 295.2670, Y 54.8727, Z -7.1667, A 0.000, B 0.000, C 0.000 }
gfCNCPoint5[18483] = {X 295.9004, Y 55.5060, Z -7.1667, A 0.000, B 0.000, C 0.000 }
gfCNCPoint5[18484] = {X 296.3770, Y 56.2645, Z -7.1667, A 0.000, B 0.000, C 0.000 }
gfCNCPoint5[18485] = {X 296.6728, Y 57.1099, Z -7.1667, A 0.000, B 0.000, C 0.000 }
gfCNCPoint5[18486] = {X 296.7731, Y 58.0000, Z -7.1667, A 0.000, B 0.000, C 0.000 }
gfCNCPoint5[18487] = {X 296.7731, Y 58.9341, Z -7.1667, A 0.000, B 0.000, C 0.000 }
gfCNCPoint5[18488] = {X 296.6602, Y 59.8686, Z -7.1667, A 0.000, B 0.000, C 0.000 }
gfCNCPoint5[18489] = {X 296.3328, Y 60.7512, Z -7.1667, A 0.000, B 0.000, C 0.000 }
gfCNCPoint5[18490] = {X 295.8090, Y 61.5334, Z -7.1667, A 0.000, B 0.000, C 0.000 }
gfCNCPoint5[18491] = {X 295.1176, Y 62.1721, Z -7.1667, A 0.000, B 0.000, C 0.000 }
gfCNCPoint5[18492] = {X 294.2964, Y 62.6323, Z -7.1667, A 0.000, B 0.000, C 0.000 }
gfCNCPoint5[18493] = {X 293.3907, Y 62.8888, Z -7.1667, A 0.000, B 0.000, C 0.000 }
gfCNCPoint5[18494] = {X 293.2333, Y 62.9107, Z -7.1667, A 0.000, B 0.000, C 0.000 }
gfCNCPoint5[18495] = {X 293.0752, Y 62.9264, Z -7.1667, A 0.000, B 0.000, C 0.000 }
gfCNCPoint5[18496] = {X 293.0538, Y 63.1540, Z -7.1667, A 0.000, B 0.000, C 0.000 }
gfCNCPoint5[18497] = {X 293.0538, Y 92.9237, Z -7.1667, A 0.000, B 0.000, C 0.000 }
gfCNCPoint5[18498] = {X 293.0752, Y 93.0661, Z -7.1667, A 0.000, B 0.000, C 0.000 }
gfCNCPoint5[18499] = {X 293.2327, Y 93.0823, Z -7.1667, A 0.000, B 0.000, C 0.000 }
gfCNCPoint5[18500] = {X 293.3894, Y 93.1047, Z -7.1667, A 0.000, B 0.000, C 0.000 }
gfCNCPoint5[18501] = {X 294.2949, Y 93.3638, Z -7.1667, A 0.000, B 0.000, C 0.000 }
gfCNCPoint5[18502] = {X 295.1157, Y 93.8258, Z -7.1667, A 0.000, B 0.000, C 0.000 }
gfCNCPoint5[18503] = {X 295.8068, Y 94.4656, Z -7.1667, A 0.000, B 0.000, C 0.000 }
gfCNCPoint5[18504] = {X 296.3307, Y 95.2483, Z -7.1667, A 0.000, B 0.000, C 0.000 }
gfCNCPoint5[18505] = {X 296.6588, Y 96.1311, Z -7.1667, A 0.000, B 0.000, C 0.000 }
gfCNCPoint5[18506] = {X 296.7731, Y 97.0660, Z -7.1667, A 0.000, B 0.000, C 0.000 }
gfCNCPoint5[18507] = {X 296.7731, Y 98.0000, Z -7.1667, A 0.000, B 0.000, C 0.000 }
gfCNCPoint5[18508] = {X 296.6728, Y 98.8901, Z -7.1667, A 0.000, B 0.000, C 0.000 }
gfCNCPoint5[18509] = {X 296.3770, Y 99.7355, Z -7.1667, A 0.000, B 0.000, C 0.000 }
gfCNCPoint5[18510] = {X 295.9004, Y 100.4940, Z -7.1667, A 0.000, B 0.000, C 0.000 }
gfCNCPoint5[18511] = {X 295.2670, Y 101.1273, Z -7.1667, A 0.000, B 0.000, C 0.000 }
gfCNCPoint5[18512] = {X 294.5086, Y 101.6039, Z -7.1667, A 0.000, B 0.000, C 0.000 }
gfCNCPoint5[18513] = {X 293.6632, Y 101.8997, Z -7.1667, A 0.000, B 0.000, C 0.000 }
gfCNCPoint5[18514] = {X 292.7731, Y 102.0000, Z -7.1667, A 0.000, B 0.000, C 0.000 }
gfCNCPoint5[18515] = {X 276.2327, Y 102.0000, Z -7.1667, A 0.000, B 0.000, C 0.000 }
gfCNCPoint5[18516] = {X 275.3426, Y 101.8997, Z -7.1667, A 0.000, B 0.000, C 0.000 }
gfCNCPoint5[18517] = {X 274.4972, Y 101.6039, Z -7.1667, A 0.000, B 0.000, C 0.000 }
gfCNCPoint5[18518] = {X 273.7387, Y 101.1273, Z -7.1667, A 0.000, B 0.000, C 0.000 }
gfCNCPoint5[18519] = {X 273.1054, Y 100.4940, Z -7.1667, A 0.000, B 0.000, C 0.000 }
gfCNCPoint5[18520] = {X 272.6288, Y 99.7355, Z -7.1667, A 0.000, B 0.000, C 0.000 }
gfCNCPoint5[18521] = {X 272.3330, Y 98.8901, Z -7.1667, A 0.000, B 0.000, C 0.000 }
gfCNCPoint5[18522] = {X 272.2327, Y 98.0000, Z -7.1667, A 0.000, B 0.000, C 0.000 }
gfCNCPoint5[18523] = {X 272.2329, Y 97.0232, Z -7.1667, A 0.000, B 0.000, C 0.000 }
gfCNCPoint5[18524] = {X 272.3321, Y 96.1797, Z -7.1667, A 0.000, B 0.000, C 0.000 }
gfCNCPoint5[18525] = {X 272.6072, Y 95.3761, Z -7.1667, A 0.000, B 0.000, C 0.000 }
gfCNCPoint5[18526] = {X 273.0457, Y 94.6486, Z -7.1667, A 0.000, B 0.000, C 0.000 }
gfCNCPoint5[18527] = {X 273.6280, Y 94.0302, Z -7.1667, A 0.000, B 0.000, C 0.000 }
gfCNCPoint5[18528] = {X 274.3277, Y 93.5487, Z -7.1667, A 0.000, B 0.000, C 0.000 }
gfCNCPoint5[18529] = {X 275.1133, Y 93.2258, Z -7.1667, A 0.000, B 0.000, C 0.000 }
gfCNCPoint5[18530] = {X 275.9494, Y 93.0760, Z -7.1667, A 0.000, B 0.000, C 0.000 }
gfCNCPoint5[18531] = {X 275.9494, Y 85.3767, Z -7.1667, A 0.000, B 0.000, C 0.000 }
gfCNCPoint5[18532] = {X 262.6059, Y 80.1460, Z -7.1667, A 0.000, B 0.000, C 0.000 }
gfCNCPoint5[18533] = {X 262.1057, Y 80.4620, Z -7.1667, A 0.000, B 0.000, C 0.000 }
gfCNCPoint5[18534] = {X 237.4765, Y 96.4149, Z -7.1667, A 0.000, B 0.000, C 0.000 }
gfCNCPoint5[18535] = {X 237.4798, Y 97.0659, Z -7.1667, A 0.000, B 0.000, C 0.000 }
gfCNCPoint5[18536] = {X 237.4798, Y 98.0000, Z -7.1667, A 0.000, B 0.000, C 0.000 }
gfCNCPoint5[18537] = {X 237.3795, Y 98.8901, Z -7.1667, A 0.000, B 0.000, C 0.000 }
gfCNCPoint5[18538] = {X 237.0837, Y 99.7355, Z -7.1667, A 0.000, B 0.000, C 0.000 }
gfCNCPoint5[18539] = {X 236.6071, Y 100.4940, Z -7.1667, A 0.000, B 0.000, C 0.000 }
gfCNCPoint5[18540] = {X 235.9737, Y 101.1273, Z -7.1667, A 0.000, B 0.000, C 0.000 }
gfCNCPoint5[18541] = {X 235.2153, Y 101.6039, Z -7.1667, A 0.000, B 0.000, C 0.000 }
gfCNCPoint5[18542] = {X 234.3699, Y 101.8997, Z -7.1667, A 0.000, B 0.000, C 0.000 }
gfCNCPoint5[18543] = {X 233.4798, Y 102.0000, Z -7.1667, A 0.000, B 0.000, C 0.000 }
gfCNCPoint5[18544] = {X 214.1790, Y 102.0000, Z -7.1667, A 0.000, B 0.000, C 0.000 }
gfCNCPoint5[18545] = {X 213.7859, Y 101.9806, Z -7.1667, A 0.000, B 0.000, C 0.000 }
gfCNCPoint5[18546] = {X 213.3966, Y 101.9227, Z -7.1667, A 0.000, B 0.000, C 0.000 }
gfCNCPoint5[18547] = {X 213.0072, Y 101.9806, Z -7.1667, A 0.000, B 0.000, C 0.000 }
gfCNCPoint5[18548] = {X 212.6141, Y 102.0000, Z -7.1667, A 0.000, B 0.000, C 0.000 }
gfCNCPoint5[18549] = {X 194.9870, Y 102.0000, Z -7.1667, A 0.000, B 0.000, C 0.000 }
gfCNCPoint5[18550] = {X 194.0969, Y 101.8997, Z -7.1667, A 0.000, B 0.000, C 0.000 }
gfCNCPoint5[18551] = {X 193.2514, Y 101.6039, Z -7.1667, A 0.000, B 0.000, C 0.000 }
gfCNCPoint5[18552] = {X 192.4930, Y 101.1273, Z -7.1667, A 0.000, B 0.000, C 0.000 }
gfCNCPoint5[18553] = {X 191.8596, Y 100.4940, Z -7.1667, A 0.000, B 0.000, C 0.000 }
gfCNCPoint5[18554] = {X 191.3831, Y 99.7355, Z -7.1667, A 0.000, B 0.000, C 0.000 }
gfCNCPoint5[18555] = {X 191.0872, Y 98.8901, Z -7.1667, A 0.000, B 0.000, C 0.000 }
gfCNCPoint5[18556] = {X 190.9870, Y 98.0000, Z -7.1667, A 0.000, B 0.000, C 0.000 }
gfCNCPoint5[18557] = {X 190.9870, Y 97.0659, Z -7.1667, A 0.000, B 0.000, C 0.000 }
gfCNCPoint5[18558] = {X 191.0804, Y 96.2066, Z -7.1667, A 0.000, B 0.000, C 0.000 }
gfCNCPoint5[18559] = {X 191.3562, Y 95.3874, Z -7.1667, A 0.000, B 0.000, C 0.000 }
gfCNCPoint5[18560] = {X 191.8015, Y 94.6466, Z -7.1667, A 0.000, B 0.000, C 0.000 }
gfCNCPoint5[18561] = {X 191.9052, Y 94.5174, Z -7.1667, A 0.000, B 0.000, C 0.000 }
gfCNCPoint5[18562] = {X 192.0142, Y 94.3925, Z -7.1667, A 0.000, B 0.000, C 0.000 }
gfCNCPoint5[18563] = {X 188.7055, Y 90.7802, Z -7.1667, A 0.000, B 0.000, C 0.000 }
gfCNCPoint5[18564] = {X 149.9476, Y 90.7802, Z -7.1667, A 0.000, B 0.000, C 0.000 }
gfCNCPoint5[18565] = {X 146.7194, Y 94.3567, Z -7.1667, A 0.000, B 0.000, C 0.000 }
gfCNCPoint5[18566] = {X 147.1696, Y 94.9479, Z -7.1667, A 0.000, B 0.000, C 0.000 }
gfCNCPoint5[18567] = {X 147.5032, Y 95.6120, Z -7.1667, A 0.000, B 0.000, C 0.000 }
gfCNCPoint5[18568] = {X 147.7087, Y 96.3262, Z -7.1667, A 0.000, B 0.000, C 0.000 }
gfCNCPoint5[18569] = {X 147.7791, Y 97.0660, Z -7.1667, A 0.000, B 0.000, C 0.000 }
gfCNCPoint5[18570] = {X 147.7791, Y 98.0000, Z -7.1667, A 0.000, B 0.000, C 0.000 }
gfCNCPoint5[18571] = {X 147.6788, Y 98.8901, Z -7.1667, A 0.000, B 0.000, C 0.000 }
gfCNCPoint5[18572] = {X 147.3830, Y 99.7355, Z -7.1667, A 0.000, B 0.000, C 0.000 }
gfCNCPoint5[18573] = {X 146.9064, Y 100.4940, Z -7.1667, A 0.000, B 0.000, C 0.000 }
gfCNCPoint5[18574] = {X 146.2731, Y 101.1273, Z -7.1667, A 0.000, B 0.000, C 0.000 }
gfCNCPoint5[18575] = {X 145.5146, Y 101.6039, Z -7.1667, A 0.000, B 0.000, C 0.000 }
gfCNCPoint5[18576] = {X 144.6692, Y 101.8997, Z -7.1667, A 0.000, B 0.000, C 0.000 }
gfCNCPoint5[18577] = {X 143.7791, Y 102.0000, Z -7.1667, A 0.000, B 0.000, C 0.000 }
gfCNCPoint5[18578] = {X 125.0000, Y 102.0000, Z -7.1667, A 0.000, B 0.000, C 0.000 }
gfCNCPoint5[18579] = {X 124.1099, Y 101.8997, Z -7.1667, A 0.000, B 0.000, C 0.000 }
gfCNCPoint5[18580] = {X 123.2645, Y 101.6039, Z -7.1667, A 0.000, B 0.000, C 0.000 }
gfCNCPoint5[18581] = {X 122.5060, Y 101.1273, Z -7.1667, A 0.000, B 0.000, C 0.000 }
gfCNCPoint5[18582] = {X 121.8727, Y 100.4940, Z -7.1667, A 0.000, B 0.000, C 0.000 }
gfCNCPoint5[18583] = {X 121.3961, Y 99.7355, Z -7.1667, A 0.000, B 0.000, C 0.000 }
gfCNCPoint5[18584] = {X 121.1003, Y 98.8901, Z -7.1667, A 0.000, B 0.000, C 0.000 }
gfCNCPoint5[18585] = {X 121.0000, Y 98.0000, Z -7.1667, A 0.000, B 0.000, C 0.000 }
gfCNCPoint5[18586] = {X 121.0000, Y 97.0659, Z -7.1667, A 0.000, B 0.000, C 0.000 }
gfCNCPoint5[18587] = {X 121.0981, Y 96.1853, Z -7.1667, A 0.000, B 0.000, C 0.000 }
gfCNCPoint5[18588] = {X 121.3877, Y 95.3479, Z -7.1667, A 0.000, B 0.000, C 0.000 }
gfCNCPoint5[18589] = {X 121.8546, Y 94.5948, Z -7.1667, A 0.000, B 0.000, C 0.000 }
gfCNCPoint5[18590] = {X 122.4758, Y 93.9629, Z -7.1667, A 0.000, B 0.000, C 0.000 }
gfCNCPoint5[18591] = {X 123.2209, Y 93.4834, Z -7.1667, A 0.000, B 0.000, C 0.000 }
gfCNCPoint5[18592] = {X 124.0533, Y 93.1796, Z -7.1667, A 0.000, B 0.000, C 0.000 }
gfCNCPoint5[18593] = {X 124.9321, Y 93.0665, Z -7.1667, A 0.000, B 0.000, C 0.000 }
gfCNCPoint5[18594] = {X 124.9747, Y 93.0370, Z -7.1667, A 0.000, B 0.000, C 0.000 }
gfCNCPoint5[18595] = {X 125.4940, Y 92.9600, Z -7.1667, A 0.000, B 0.000, C 0.000 }
gfCNCPoint5[18596] = {X 126.3821, Y 92.8091, Z -7.1667, A 0.000, B 0.000, C 0.000 }
gfCNCPoint5[18597] = {X 127.2572, Y 92.5952, Z -7.1667, A 0.000, B 0.000, C 0.000 }
gfCNCPoint5[18598] = {X 128.4862, Y 91.4440, Z -7.1667, A 0.000, B 0.000, C 0.000 }
gfCNCPoint5[18599] = {X 129.6489, Y 90.2259, Z -7.1667, A 0.000, B 0.000, C 0.000 }
gfCNCPoint5[18600] = {X 140.9160, Y 77.8539, Z -7.1667, A 0.000, B 0.000, C 0.000 }
gfCNCPoint5[18601] = {X 137.8994, Y 75.1068, Z -7.1667, A 0.000, B 0.000, C 0.000 }
gfCNCPoint5[18602] = {X 137.8994, Y 75.1068, Z -4.1667, A 0.000, B 0.000, C 0.000 }
gfCNCPoint5[18603] = {X 137.8994, Y 75.1068, Z 11.0000, A 0.000, B 0.000, C 0.000 }
gfCNCPoint5[18604] = {X 165.2861, Y 38.5771, Z 11.0000, A 0.000, B 0.000, C 0.000 }
gfCNCPoint5[18605] = {X 165.2861, Y 38.5771, Z -4.1667, A 0.000, B 0.000, C 0.000 }
gfCNCPoint5[18606] = {X 165.2861, Y 38.5771, Z -7.1667, A 0.000, B 0.000, C 0.000 }
gfCNCPoint5[18607] = {X 169.3153, Y 37.9356, Z -7.1667, A 0.000, B 0.000, C 0.000 }
gfCNCPoint5[18608] = {X 169.2598, Y 37.5869, Z -7.1667, A 0.000, B 0.000, C 0.000 }
gfCNCPoint5[18609] = {X 169.1017, Y 35.9822, Z -7.1667, A 0.000, B 0.000, C 0.000 }
gfCNCPoint5[18610] = {X 169.1189, Y 34.3699, Z -7.1667, A 0.000, B 0.000, C 0.000 }
gfCNCPoint5[18611] = {X 169.3111, Y 32.7690, Z -7.1667, A 0.000, B 0.000, C 0.000 }
gfCNCPoint5[18612] = {X 169.6761, Y 31.1984, Z -7.1667, A 0.000, B 0.000, C 0.000 }
gfCNCPoint5[18613] = {X 170.2094, Y 29.6767, Z -7.1667, A 0.000, B 0.000, C 0.000 }
gfCNCPoint5[18614] = {X 170.8481, Y 28.3698, Z -7.1667, A 0.000, B 0.000, C 0.000 }
gfCNCPoint5[18615] = {X 171.6557, Y 27.1600, Z -7.1667, A 0.000, B 0.000, C 0.000 }
gfCNCPoint5[18616] = {X 172.6179, Y 26.0690, Z -7.1667, A 0.000, B 0.000, C 0.000 }
gfCNCPoint5[18617] = {X 173.7173, Y 25.1165, Z -7.1667, A 0.000, B 0.000, C 0.000 }
gfCNCPoint5[18618] = {X 174.9342, Y 24.3196, Z -7.1667, A 0.000, B 0.000, C 0.000 }
gfCNCPoint5[18619] = {X 174.1518, Y 23.9320, Z -7.1667, A 0.000, B 0.000, C 0.000 }
gfCNCPoint5[18620] = {X 173.4634, Y 23.3949, Z -7.1667, A 0.000, B 0.000, C 0.000 }
gfCNCPoint5[18621] = {X 172.8970, Y 22.7303, Z -7.1667, A 0.000, B 0.000, C 0.000 }
gfCNCPoint5[18622] = {X 172.4758, Y 21.9655, Z -7.1667, A 0.000, B 0.000, C 0.000 }
gfCNCPoint5[18623] = {X 169.8405, Y 15.5121, Z -7.1667, A 0.000, B 0.000, C 0.000 }
gfCNCPoint5[18624] = {X 169.5912, Y 14.6607, Z -7.1667, A 0.000, B 0.000, C 0.000 }
gfCNCPoint5[18625] = {X 169.5212, Y 13.7764, Z -7.1667, A 0.000, B 0.000, C 0.000 }
gfCNCPoint5[18626] = {X 169.6332, Y 12.8964, Z -7.1667, A 0.000, B 0.000, C 0.000 }
gfCNCPoint5[18627] = {X 169.9226, Y 12.0578, Z -7.1667, A 0.000, B 0.000, C 0.000 }
gfCNCPoint5[18628] = {X 170.3773, Y 11.2960, Z -7.1667, A 0.000, B 0.000, C 0.000 }
gfCNCPoint5[18629] = {X 170.9779, Y 10.6432, Z -7.1667, A 0.000, B 0.000, C 0.000 }
gfCNCPoint5[18630] = {X 171.6992, Y 10.1268, Z -7.1667, A 0.000, B 0.000, C 0.000 }
gfCNCPoint5[18631] = {X 172.3295, Y 9.7674, Z -7.1667, A 0.000, B 0.000, C 0.000 }
gfCNCPoint5[18632] = {X 173.1919, Y 9.4018, Z -7.1667, A 0.000, B 0.000, C 0.000 }
gfCNCPoint5[18633] = {X 174.1128, Y 9.2306, Z -7.1667, A 0.000, B 0.000, C 0.000 }
gfCNCPoint5[18634] = {X 175.0490, Y 9.2620, Z -7.1667, A 0.000, B 0.000, C 0.000 }
gfCNCPoint5[18635] = {X 175.9563, Y 9.4944, Z -7.1667, A 0.000, B 0.000, C 0.000 }
gfCNCPoint5[18636] = {X 177.1291, Y 9.0434, Z -7.1667, A 0.000, B 0.000, C 0.000 }
gfCNCPoint5[18637] = {X 179.2988, Y 8.2449, Z -7.1667, A 0.000, B 0.000, C 0.000 }
gfCNCPoint5[18638] = {X 181.5367, Y 7.6643, Z -7.1667, A 0.000, B 0.000, C 0.000 }
gfCNCPoint5[18639] = {X 183.8210, Y 7.3074, Z -7.1667, A 0.000, B 0.000, C 0.000 }
gfCNCPoint5[18640] = {X 186.1293, Y 7.1775, Z -7.1667, A 0.000, B 0.000, C 0.000 }
gfCNCPoint5[18641] = {X 188.4392, Y 7.2760, Z -7.1667, A 0.000, B 0.000, C 0.000 }
gfCNCPoint5[18642] = {X 190.7281, Y 7.6019, Z -7.1667, A 0.000, B 0.000, C 0.000 }
gfCNCPoint5[18643] = {X 192.3169, Y 7.9885, Z -7.1667, A 0.000, B 0.000, C 0.000 }
gfCNCPoint5[18644] = {X 193.8616, Y 8.5251, Z -7.1667, A 0.000, B 0.000, C 0.000 }
gfCNCPoint5[18645] = {X 195.3479, Y 9.2067, Z -7.1667, A 0.000, B 0.000, C 0.000 }
gfCNCPoint5[18646] = {X 196.7623, Y 10.0273, Z -7.1667, A 0.000, B 0.000, C 0.000 }
gfCNCPoint5[18647] = {X 198.0919, Y 10.9792, Z -7.1667, A 0.000, B 0.000, C 0.000 }
gfCNCPoint5[18648] = {X 199.1517, Y 11.9221, Z -7.1667, A 0.000, B 0.000, C 0.000 }
gfCNCPoint5[18649] = {X 200.1027, Y 12.9747, Z -7.1667, A 0.000, B 0.000, C 0.000 }
gfCNCPoint5[18650] = {X 200.9335, Y 14.1244, Z -7.1667, A 0.000, B 0.000, C 0.000 }
gfCNCPoint5[18651] = {X 201.6344, Y 15.3577, Z -7.1667, A 0.000, B 0.000, C 0.000 }
gfCNCPoint5[18652] = {X 202.1970, Y 16.6600, Z -7.1667, A 0.000, B 0.000, C 0.000 }
gfCNCPoint5[18653] = {X 202.6712, Y 18.3163, Z -7.1667, A 0.000, B 0.000, C 0.000 }
gfCNCPoint5[18654] = {X 202.9527, Y 20.0160, Z -7.1667, A 0.000, B 0.000, C 0.000 }
gfCNCPoint5[18655] = {X 203.0377, Y 21.7368, Z -7.1667, A 0.000, B 0.000, C 0.000 }
gfCNCPoint5[18656] = {X 202.9251, Y 23.4560, Z -7.1667, A 0.000, B 0.000, C 0.000 }
gfCNCPoint5[18657] = {X 202.6165, Y 25.1510, Z -7.1667, A 0.000, B 0.000, C 0.000 }
gfCNCPoint5[18658] = {X 202.1745, Y 26.5972, Z -7.1667, A 0.000, B 0.000, C 0.000 }
gfCNCPoint5[18659] = {X 201.5497, Y 27.9742, Z -7.1667, A 0.000, B 0.000, C 0.000 }
gfCNCPoint5[18660] = {X 200.7525, Y 29.2592, Z -7.1667, A 0.000, B 0.000, C 0.000 }
gfCNCPoint5[18661] = {X 199.7961, Y 30.4305, Z -7.1667, A 0.000, B 0.000, C 0.000 }
gfCNCPoint5[18662] = {X 198.6966, Y 31.4687, Z -7.1667, A 0.000, B 0.000, C 0.000 }
gfCNCPoint5[18663] = {X 199.4976, Y 31.8099, Z -7.1667, A 0.000, B 0.000, C 0.000 }
gfCNCPoint5[18664] = {X 200.2138, Y 32.3048, Z -7.1667, A 0.000, B 0.000, C 0.000 }
gfCNCPoint5[18665] = {X 200.8163, Y 32.9333, Z -7.1667, A 0.000, B 0.000, C 0.000 }
gfCNCPoint5[18666] = {X 201.2806, Y 33.6698, Z -7.1667, A 0.000, B 0.000, C 0.000 }
gfCNCPoint5[18667] = {X 204.3222, Y 39.9530, Z -7.1667, A 0.000, B 0.000, C 0.000 }
gfCNCPoint5[18668] = {X 204.6427, Y 40.8622, Z -7.1667, A 0.000, B 0.000, C 0.000 }
gfCNCPoint5[18669] = {X 204.7537, Y 41.8197, Z -7.1667, A 0.000, B 0.000, C 0.000 }
gfCNCPoint5[18670] = {X 204.6496, Y 42.7781, Z -7.1667, A 0.000, B 0.000, C 0.000 }
gfCNCPoint5[18671] = {X 204.3355, Y 43.6895, Z -7.1667, A 0.000, B 0.000, C 0.000 }
gfCNCPoint5[18672] = {X 203.8272, Y 44.5085, Z -7.1667, A 0.000, B 0.000, C 0.000 }
gfCNCPoint5[18673] = {X 203.1499, Y 45.1945, Z -7.1667, A 0.000, B 0.000, C 0.000 }
gfCNCPoint5[18674] = {X 202.6137, Y 45.6280, Z -7.1667, A 0.000, B 0.000, C 0.000 }
gfCNCPoint5[18675] = {X 201.9093, Y 46.0919, Z -7.1667, A 0.000, B 0.000, C 0.000 }
gfCNCPoint5[18676] = {X 201.1283, Y 46.4105, Z -7.1667, A 0.000, B 0.000, C 0.000 }
gfCNCPoint5[18677] = {X 200.3003, Y 46.5718, Z -7.1667, A 0.000, B 0.000, C 0.000 }
gfCNCPoint5[18678] = {X 199.4569, Y 46.5697, Z -7.1667, A 0.000, B 0.000, C 0.000 }
gfCNCPoint5[18679] = {X 198.6298, Y 46.4041, Z -7.1667, A 0.000, B 0.000, C 0.000 }
gfCNCPoint5[18680] = {X 196.5192, Y 47.5050, Z -7.1667, A 0.000, B 0.000, C 0.000 }
gfCNCPoint5[18681] = {X 194.3239, Y 48.4254, Z -7.1667, A 0.000, B 0.000, C 0.000 }
gfCNCPoint5[18682] = {X 192.0593, Y 49.1589, Z -7.1667, A 0.000, B 0.000, C 0.000 }
gfCNCPoint5[18683] = {X 189.8462, Y 49.6714, Z -7.1667, A 0.000, B 0.000, C 0.000 }
gfCNCPoint5[18684] = {X 187.5926, Y 49.9573, Z -7.1667, A 0.000, B 0.000, C 0.000 }
gfCNCPoint5[18685] = {X 185.3216, Y 50.0135, Z -7.1667, A 0.000, B 0.000, C 0.000 }
gfCNCPoint5[18686] = {X 183.0566, Y 49.8396, Z -7.1667, A 0.000, B 0.000, C 0.000 }
gfCNCPoint5[18687] = {X 180.8208, Y 49.4372, Z -7.1667, A 0.000, B 0.000, C 0.000 }
gfCNCPoint5[18688] = {X 178.9806, Y 48.9038, Z -7.1667, A 0.000, B 0.000, C 0.000 }
gfCNCPoint5[18689] = {X 177.2142, Y 48.1618, Z -7.1667, A 0.000, B 0.000, C 0.000 }
gfCNCPoint5[18690] = {X 175.5450, Y 47.2211, Z -7.1667, A 0.000, B 0.000, C 0.000 }
gfCNCPoint5[18691] = {X 173.9955, Y 46.0942, Z -7.1667, A 0.000, B 0.000, C 0.000 }
gfCNCPoint5[18692] = {X 172.8548, Y 45.0533, Z -7.1667, A 0.000, B 0.000, C 0.000 }
gfCNCPoint5[18693] = {X 171.8452, Y 43.8848, Z -7.1667, A 0.000, B 0.000, C 0.000 }
gfCNCPoint5[18694] = {X 170.9810, Y 42.6050, Z -7.1667, A 0.000, B 0.000, C 0.000 }
gfCNCPoint5[18695] = {X 170.2743, Y 41.2320, Z -7.1667, A 0.000, B 0.000, C 0.000 }
gfCNCPoint5[18696] = {X 169.7351, Y 39.7849, Z -7.1667, A 0.000, B 0.000, C 0.000 }
gfCNCPoint5[18697] = {X 169.3708, Y 38.2842, Z -7.1667, A 0.000, B 0.000, C 0.000 }
gfCNCPoint5[18698] = {X 169.3153, Y 37.9356, Z -7.1667, A 0.000, B 0.000, C 0.000 }
gfCNCPoint5[18699] = {X 165.3651, Y 38.5645, Z -7.1667, A 0.000, B 0.000, C 0.000 }
gfCNCPoint5[18700] = {X 169.3943, Y 37.9230, Z -7.1667, A 0.000, B 0.000, C 0.000 }
gfCNCPoint5[18701] = {X 169.3389, Y 37.5748, Z -7.1667, A 0.000, B 0.000, C 0.000 }
gfCNCPoint5[18702] = {X 169.1817, Y 35.9787, Z -7.1667, A 0.000, B 0.000, C 0.000 }
gfCNCPoint5[18703] = {X 169.1987, Y 34.3750, Z -7.1667, A 0.000, B 0.000, C 0.000 }
gfCNCPoint5[18704] = {X 169.3899, Y 32.7827, Z -7.1667, A 0.000, B 0.000, C 0.000 }
gfCNCPoint5[18705] = {X 169.7529, Y 31.2205, Z -7.1667, A 0.000, B 0.000, C 0.000 }
gfCNCPoint5[18706] = {X 170.2835, Y 29.7070, Z -7.1667, A 0.000, B 0.000, C 0.000 }
gfCNCPoint5[18707] = {X 170.9351, Y 28.3789, Z -7.1667, A 0.000, B 0.000, C 0.000 }
gfCNCPoint5[18708] = {X 171.7626, Y 27.1525, Z -7.1667, A 0.000, B 0.000, C 0.000 }
gfCNCPoint5[18709] = {X 172.7503, Y 26.0511, Z -7.1667, A 0.000, B 0.000, C 0.000 }
gfCNCPoint5[18710] = {X 173.8796, Y 25.0954, Z -7.1667, A 0.000, B 0.000, C 0.000 }
gfCNCPoint5[18711] = {X 175.1292, Y 24.3034, Z -7.1667, A 0.000, B 0.000, C 0.000 }
gfCNCPoint5[18712] = {X 174.3079, Y 23.9332, Z -7.1667, A 0.000, B 0.000, C 0.000 }
gfCNCPoint5[18713] = {X 173.5834, Y 23.3978, Z -7.1667, A 0.000, B 0.000, C 0.000 }
gfCNCPoint5[18714] = {X 172.9884, Y 22.7215, Z -7.1667, A 0.000, B 0.000, C 0.000 }
gfCNCPoint5[18715] = {X 172.5496, Y 21.9347, Z -7.1667, A 0.000, B 0.000, C 0.000 }
gfCNCPoint5[18716] = {X 169.9145, Y 15.4818, Z -7.1667, A 0.000, B 0.000, C 0.000 }
gfCNCPoint5[18717] = {X 169.6699, Y 14.6462, Z -7.1667, A 0.000, B 0.000, C 0.000 }
gfCNCPoint5[18718] = {X 169.6011, Y 13.7783, Z -7.1667, A 0.000, B 0.000, C 0.000 }
gfCNCPoint5[18719] = {X 169.7111, Y 12.9146, Z -7.1667, A 0.000, B 0.000, C 0.000 }
gfCNCPoint5[18720] = {X 169.9952, Y 12.0915, Z -7.1667, A 0.000, B 0.000, C 0.000 }
gfCNCPoint5[18721] = {X 170.4414, Y 11.3439, Z -7.1667, A 0.000, B 0.000, C 0.000 }
gfCNCPoint5[18722] = {X 171.0309, Y 10.7031, Z -7.1667, A 0.000, B 0.000, C 0.000 }
gfCNCPoint5[18723] = {X 171.7389, Y 10.1963, Z -7.1667, A 0.000, B 0.000, C 0.000 }
gfCNCPoint5[18724] = {X 172.3689, Y 9.8371, Z -7.1667, A 0.000, B 0.000, C 0.000 }
gfCNCPoint5[18725] = {X 173.2225, Y 9.4762, Z -7.1667, A 0.000, B 0.000, C 0.000 }
gfCNCPoint5[18726] = {X 174.1341, Y 9.3093, Z -7.1667, A 0.000, B 0.000, C 0.000 }
gfCNCPoint5[18727] = {X 175.0602, Y 9.3445, Z -7.1667, A 0.000, B 0.000, C 0.000 }
gfCNCPoint5[18728] = {X 175.9565, Y 9.5801, Z -7.1667, A 0.000, B 0.000, C 0.000 }
gfCNCPoint5[18729] = {X 177.1591, Y 9.1175, Z -7.1667, A 0.000, B 0.000, C 0.000 }
gfCNCPoint5[18730] = {X 179.3216, Y 8.3216, Z -7.1667, A 0.000, B 0.000, C 0.000 }
gfCNCPoint5[18731] = {X 181.5520, Y 7.7429, Z -7.1667, A 0.000, B 0.000, C 0.000 }
gfCNCPoint5[18732] = {X 183.8287, Y 7.3870, Z -7.1667, A 0.000, B 0.000, C 0.000 }
gfCNCPoint5[18733] = {X 186.1294, Y 7.2575, Z -7.1667, A 0.000, B 0.000, C 0.000 }
gfCNCPoint5[18734] = {X 188.4316, Y 7.3557, Z -7.1667, A 0.000, B 0.000, C 0.000 }
gfCNCPoint5[18735] = {X 190.7129, Y 7.6805, Z -7.1667, A 0.000, B 0.000, C 0.000 }
gfCNCPoint5[18736] = {X 192.2943, Y 8.0652, Z -7.1667, A 0.000, B 0.000, C 0.000 }
gfCNCPoint5[18737] = {X 193.8317, Y 8.5993, Z -7.1667, A 0.000, B 0.000, C 0.000 }
gfCNCPoint5[18738] = {X 195.3111, Y 9.2778, Z -7.1667, A 0.000, B 0.000, C 0.000 }
gfCNCPoint5[18739] = {X 196.7189, Y 10.0945, Z -7.1667, A 0.000, B 0.000, C 0.000 }
gfCNCPoint5[18740] = {X 198.0422, Y 11.0420, Z -7.1667, A 0.000, B 0.000, C 0.000 }
gfCNCPoint5[18741] = {X 199.0955, Y 11.9790, Z -7.1667, A 0.000, B 0.000, C 0.000 }
gfCNCPoint5[18742] = {X 200.0406, Y 13.0251, Z -7.1667, A 0.000, B 0.000, C 0.000 }
gfCNCPoint5[18743] = {X 200.8663, Y 14.1678, Z -7.1667, A 0.000, B 0.000, C 0.000 }
gfCNCPoint5[18744] = {X 201.5629, Y 15.3935, Z -7.1667, A 0.000, B 0.000, C 0.000 }
gfCNCPoint5[18745] = {X 202.1220, Y 16.6876, Z -7.1667, A 0.000, B 0.000, C 0.000 }
gfCNCPoint5[18746] = {X 202.5935, Y 18.3350, Z -7.1667, A 0.000, B 0.000, C 0.000 }
gfCNCPoint5[18747] = {X 202.8733, Y 20.0254, Z -7.1667, A 0.000, B 0.000, C 0.000 }
gfCNCPoint5[18748] = {X 202.9577, Y 21.7368, Z -7.1667, A 0.000, B 0.000, C 0.000 }
gfCNCPoint5[18749] = {X 202.8457, Y 23.4467, Z -7.1667, A 0.000, B 0.000, C 0.000 }
gfCNCPoint5[18750] = {X 202.5386, Y 25.1324, Z -7.1667, A 0.000, B 0.000, C 0.000 }
gfCNCPoint5[18751] = {X 202.0890, Y 26.5970, Z -7.1667, A 0.000, B 0.000, C 0.000 }
gfCNCPoint5[18752] = {X 201.4506, Y 27.9897, Z -7.1667, A 0.000, B 0.000, C 0.000 }
gfCNCPoint5[18753] = {X 200.6344, Y 29.2863, Z -7.1667, A 0.000, B 0.000, C 0.000 }
gfCNCPoint5[18754] = {X 199.6547, Y 30.4642, Z -7.1667, A 0.000, B 0.000, C 0.000 }
gfCNCPoint5[18755] = {X 198.5284, Y 31.5029, Z -7.1667, A 0.000, B 0.000, C 0.000 }
gfCNCPoint5[18756] = {X 199.3594, Y 31.8268, Z -7.1667, A 0.000, B 0.000, C 0.000 }
gfCNCPoint5[18757] = {X 200.1043, Y 32.3174, Z -7.1667, A 0.000, B 0.000, C 0.000 }
gfCNCPoint5[18758] = {X 200.7300, Y 32.9530, Z -7.1667, A 0.000, B 0.000, C 0.000 }
gfCNCPoint5[18759] = {X 201.2090, Y 33.7054, Z -7.1667, A 0.000, B 0.000, C 0.000 }
gfCNCPoint5[18760] = {X 204.2502, Y 39.9879, Z -7.1667, A 0.000, B 0.000, C 0.000 }
gfCNCPoint5[18761] = {X 204.5648, Y 40.8802, Z -7.1667, A 0.000, B 0.000, C 0.000 }
gfCNCPoint5[18762] = {X 204.6737, Y 41.8200, Z -7.1667, A 0.000, B 0.000, C 0.000 }
gfCNCPoint5[18763] = {X 204.5715, Y 42.7606, Z -7.1667, A 0.000, B 0.000, C 0.000 }
gfCNCPoint5[18764] = {X 204.2633, Y 43.6551, Z -7.1667, A 0.000, B 0.000, C 0.000 }
gfCNCPoint5[18765] = {X 203.7643, Y 44.4590, Z -7.1667, A 0.000, B 0.000, C 0.000 }
gfCNCPoint5[18766] = {X 203.0996, Y 45.1323, Z -7.1667, A 0.000, B 0.000, C 0.000 }
gfCNCPoint5[18767] = {X 202.5634, Y 45.5658, Z -7.1667, A 0.000, B 0.000, C 0.000 }
gfCNCPoint5[18768] = {X 201.8659, Y 46.0243, Z -7.1667, A 0.000, B 0.000, C 0.000 }
gfCNCPoint5[18769] = {X 201.0921, Y 46.3378, Z -7.1667, A 0.000, B 0.000, C 0.000 }
gfCNCPoint5[18770] = {X 200.2721, Y 46.4941, Z -7.1667, A 0.000, B 0.000, C 0.000 }
gfCNCPoint5[18771] = {X 199.4373, Y 46.4872, Z -7.1667, A 0.000, B 0.000, C 0.000 }
gfCNCPoint5[18772] = {X 198.6200, Y 46.3174, Z -7.1667, A 0.000, B 0.000, C 0.000 }
gfCNCPoint5[18773] = {X 196.5061, Y 47.4227, Z -7.1667, A 0.000, B 0.000, C 0.000 }
gfCNCPoint5[18774] = {X 194.3068, Y 48.3464, Z -7.1667, A 0.000, B 0.000, C 0.000 }
gfCNCPoint5[18775] = {X 192.0376, Y 49.0819, Z -7.1667, A 0.000, B 0.000, C 0.000 }
gfCNCPoint5[18776] = {X 189.8323, Y 49.5926, Z -7.1667, A 0.000, B 0.000, C 0.000 }
gfCNCPoint5[18777] = {X 187.5867, Y 49.8775, Z -7.1667, A 0.000, B 0.000, C 0.000 }
gfCNCPoint5[18778] = {X 185.3237, Y 49.9335, Z -7.1667, A 0.000, B 0.000, C 0.000 }
gfCNCPoint5[18779] = {X 183.0667, Y 49.7602, Z -7.1667, A 0.000, B 0.000, C 0.000 }
gfCNCPoint5[18780] = {X 180.8388, Y 49.3592, Z -7.1667, A 0.000, B 0.000, C 0.000 }
gfCNCPoint5[18781] = {X 179.0073, Y 48.8284, Z -7.1667, A 0.000, B 0.000, C 0.000 }
gfCNCPoint5[18782] = {X 177.2493, Y 48.0899, Z -7.1667, A 0.000, B 0.000, C 0.000 }
gfCNCPoint5[18783] = {X 175.5882, Y 47.1537, Z -7.1667, A 0.000, B 0.000, C 0.000 }
gfCNCPoint5[18784] = {X 174.0460, Y 46.0322, Z -7.1667, A 0.000, B 0.000, C 0.000 }
gfCNCPoint5[18785] = {X 172.9123, Y 44.9978, Z -7.1667, A 0.000, B 0.000, C 0.000 }
gfCNCPoint5[18786] = {X 171.9090, Y 43.8365, Z -7.1667, A 0.000, B 0.000, C 0.000 }
gfCNCPoint5[18787] = {X 171.0501, Y 42.5647, Z -7.1667, A 0.000, B 0.000, C 0.000 }
gfCNCPoint5[18788] = {X 170.3477, Y 41.2002, Z -7.1667, A 0.000, B 0.000, C 0.000 }
gfCNCPoint5[18789] = {X 169.8118, Y 39.7622, Z -7.1667, A 0.000, B 0.000, C 0.000 }
gfCNCPoint5[18790] = {X 169.4497, Y 38.2708, Z -7.1667, A 0.000, B 0.000, C 0.000 }
gfCNCPoint5[18791] = {X 169.3943, Y 37.9230, Z -7.1667, A 0.000, B 0.000, C 0.000 }
gfCNCPoint5[18792] = {X 165.4441, Y 38.5519, Z -7.1667, A 0.000, B 0.000, C 0.000 }
gfCNCPoint5[18793] = {X 169.4733, Y 37.9104, Z -7.1667, A 0.000, B 0.000, C 0.000 }
gfCNCPoint5[18794] = {X 169.4179, Y 37.5626, Z -7.1667, A 0.000, B 0.000, C 0.000 }
gfCNCPoint5[18795] = {X 169.2616, Y 35.9752, Z -7.1667, A 0.000, B 0.000, C 0.000 }
gfCNCPoint5[18796] = {X 169.2786, Y 34.3801, Z -7.1667, A 0.000, B 0.000, C 0.000 }
gfCNCPoint5[18797] = {X 169.4687, Y 32.7964, Z -7.1667, A 0.000, B 0.000, C 0.000 }
gfCNCPoint5[18798] = {X 169.8298, Y 31.2427, Z -7.1667, A 0.000, B 0.000, C 0.000 }
gfCNCPoint5[18799] = {X 170.3575, Y 29.7374, Z -7.1667, A 0.000, B 0.000, C 0.000 }
gfCNCPoint5[18800] = {X 171.0238, Y 28.3856, Z -7.1667, A 0.000, B 0.000, C 0.000 }
gfCNCPoint5[18801] = {X 171.8735, Y 27.1409, Z -7.1667, A 0.000, B 0.000, C 0.000 }
gfCNCPoint5[18802] = {X 172.8898, Y 26.0280, Z -7.1667, A 0.000, B 0.000, C 0.000 }
gfCNCPoint5[18803] = {X 174.0524, Y 25.0691, Z -7.1667, A 0.000, B 0.000, C 0.000 }
gfCNCPoint5[18804] = {X 175.3383, Y 24.2831, Z -7.1667, A 0.000, B 0.000, C 0.000 }
gfCNCPoint5[18805] = {X 174.4743, Y 23.9350, Z -7.1667, A 0.000, B 0.000, C 0.000 }
gfCNCPoint5[18806] = {X 173.7094, Y 23.4033, Z -7.1667, A 0.000, B 0.000, C 0.000 }
gfCNCPoint5[18807] = {X 173.0820, Y 22.7148, Z -7.1667, A 0.000, B 0.000, C 0.000 }
gfCNCPoint5[18808] = {X 172.6235, Y 21.9039, Z -7.1667, A 0.000, B 0.000, C 0.000 }
gfCNCPoint5[18809] = {X 169.9886, Y 15.4516, Z -7.1667, A 0.000, B 0.000, C 0.000 }
gfCNCPoint5[18810] = {X 169.7252, Y 14.4911, Z -7.1667, A 0.000, B 0.000, C 0.000 }
gfCNCPoint5[18811] = {X 169.6977, Y 13.4954, Z -7.1667, A 0.000, B 0.000, C 0.000 }
gfCNCPoint5[18812] = {X 169.9076, Y 12.5218, Z -7.1667, A 0.000, B 0.000, C 0.000 }
gfCNCPoint5[18813] = {X 170.3429, Y 11.6260, Z -7.1667, A 0.000, B 0.000, C 0.000 }
gfCNCPoint5[18814] = {X 170.9787, Y 10.8594, Z -7.1667, A 0.000, B 0.000, C 0.000 }
gfCNCPoint5[18815] = {X 171.7785, Y 10.2658, Z -7.1667, A 0.000, B 0.000, C 0.000 }
gfCNCPoint5[18816] = {X 172.4082, Y 9.9068, Z -7.1667, A 0.000, B 0.000, C 0.000 }
gfCNCPoint5[18817] = {X 173.2456, Y 9.5527, Z -7.1667, A 0.000, B 0.000, C 0.000 }
gfCNCPoint5[18818] = {X 174.1400, Y 9.3891, Z -7.1667, A 0.000, B 0.000, C 0.000 }
gfCNCPoint5[18819] = {X 175.0485, Y 9.4236, Z -7.1667, A 0.000, B 0.000, C 0.000 }
gfCNCPoint5[18820] = {X 175.9279, Y 9.6548, Z -7.1667, A 0.000, B 0.000, C 0.000 }
gfCNCPoint5[18821] = {X 176.0170, Y 9.6902, Z -7.1667, A 0.000, B 0.000, C 0.000 }
gfCNCPoint5[18822] = {X 177.1904, Y 9.1912, Z -7.1667, A 0.000, B 0.000, C 0.000 }
gfCNCPoint5[18823] = {X 179.3455, Y 8.3979, Z -7.1667, A 0.000, B 0.000, C 0.000 }
gfCNCPoint5[18824] = {X 181.5683, Y 7.8212, Z -7.1667, A 0.000, B 0.000, C 0.000 }
gfCNCPoint5[18825] = {X 183.8371, Y 7.4666, Z -7.1667, A 0.000, B 0.000, C 0.000 }
gfCNCPoint5[18826] = {X 186.1299, Y 7.3375, Z -7.1667, A 0.000, B 0.000, C 0.000 }
gfCNCPoint5[18827] = {X 188.4242, Y 7.4353, Z -7.1667, A 0.000, B 0.000, C 0.000 }
gfCNCPoint5[18828] = {X 190.6977, Y 7.7590, Z -7.1667, A 0.000, B 0.000, C 0.000 }
gfCNCPoint5[18829] = {X 192.2717, Y 8.1420, Z -7.1667, A 0.000, B 0.000, C 0.000 }
gfCNCPoint5[18830] = {X 193.8019, Y 8.6735, Z -7.1667, A 0.000, B 0.000, C 0.000 }
gfCNCPoint5[18831] = {X 195.2743, Y 9.3488, Z -7.1667, A 0.000, B 0.000, C 0.000 }
gfCNCPoint5[18832] = {X 196.6755, Y 10.1617, Z -7.1667, A 0.000, B 0.000, C 0.000 }
gfCNCPoint5[18833] = {X 197.9926, Y 11.1047, Z -7.1667, A 0.000, B 0.000, C 0.000 }
gfCNCPoint5[18834] = {X 199.2845, Y 12.2861, Z -7.1667, A 0.000, B 0.000, C 0.000 }
gfCNCPoint5[18835] = {X 200.4041, Y 13.6319, Z -7.1667, A 0.000, B 0.000, C 0.000 }
gfCNCPoint5[18836] = {X 201.3305, Y 15.1173, Z -7.1667, A 0.000, B 0.000, C 0.000 }
gfCNCPoint5[18837] = {X 202.0467, Y 16.7147, Z -7.1667, A 0.000, B 0.000, C 0.000 }
gfCNCPoint5[18838] = {X 202.5155, Y 18.3531, Z -7.1667, A 0.000, B 0.000, C 0.000 }
gfCNCPoint5[18839] = {X 202.7938, Y 20.0344, Z -7.1667, A 0.000, B 0.000, C 0.000 }
gfCNCPoint5[18840] = {X 202.8777, Y 21.7366, Z -7.1667, A 0.000, B 0.000, C 0.000 }
gfCNCPoint5[18841] = {X 202.7662, Y 23.4371, Z -7.1667, A 0.000, B 0.000, C 0.000 }
gfCNCPoint5[18842] = {X 202.4608, Y 25.1138, Z -7.1667, A 0.000, B 0.000, C 0.000 }
gfCNCPoint5[18843] = {X 202.0028, Y 26.5984, Z -7.1667, A 0.000, B 0.000, C 0.000 }
gfCNCPoint5[18844] = {X 201.3495, Y 28.0081, Z -7.1667, A 0.000, B 0.000, C 0.000 }
gfCNCPoint5[18845] = {X 200.5126, Y 29.3172, Z -7.1667, A 0.000, B 0.000, C 0.000 }
gfCNCPoint5[18846] = {X 199.5074, Y 30.5020, Z -7.1667, A 0.000, B 0.000, C 0.000 }
gfCNCPoint5[18847] = {X 198.3521, Y 31.5409, Z -7.1667, A 0.000, B 0.000, C 0.000 }
gfCNCPoint5[18848] = {X 199.2152, Y 31.8443, Z -7.1667, A 0.000, B 0.000, C 0.000 }
gfCNCPoint5[18849] = {X 199.9911, Y 32.3290, Z -7.1667, A 0.000, B 0.000, C 0.000 }
gfCNCPoint5[18850] = {X 200.6423, Y 32.9716, Z -7.1667, A 0.000, B 0.000, C 0.000 }
gfCNCPoint5[18851] = {X 201.1373, Y 33.7410, Z -7.1667, A 0.000, B 0.000, C 0.000 }
gfCNCPoint5[18852] = {X 204.1781, Y 40.0227, Z -7.1667, A 0.000, B 0.000, C 0.000 }
gfCNCPoint5[18853] = {X 204.4868, Y 40.8982, Z -7.1667, A 0.000, B 0.000, C 0.000 }
gfCNCPoint5[18854] = {X 204.5937, Y 41.8203, Z -7.1667, A 0.000, B 0.000, C 0.000 }
gfCNCPoint5[18855] = {X 204.4934, Y 42.7431, Z -7.1667, A 0.000, B 0.000, C 0.000 }
gfCNCPoint5[18856] = {X 204.1910, Y 43.6208, Z -7.1667, A 0.000, B 0.000, C 0.000 }
gfCNCPoint5[18857] = {X 203.7015, Y 44.4095, Z -7.1667, A 0.000, B 0.000, C 0.000 }
gfCNCPoint5[18858] = {X 203.0493, Y 45.0700, Z -7.1667, A 0.000, B 0.000, C 0.000 }
gfCNCPoint5[18859] = {X 202.5131, Y 45.5036, Z -7.1667, A 0.000, B 0.000, C 0.000 }
gfCNCPoint5[18860] = {X 201.8225, Y 45.9567, Z -7.1667, A 0.000, B 0.000, C 0.000 }
gfCNCPoint5[18861] = {X 201.0561, Y 46.2650, Z -7.1667, A 0.000, B 0.000, C 0.000 }
gfCNCPoint5[18862] = {X 200.2440, Y 46.4163, Z -7.1667, A 0.000, B 0.000, C 0.000 }
gfCNCPoint5[18863] = {X 199.4180, Y 46.4046, Z -7.1667, A 0.000, B 0.000, C 0.000 }
gfCNCPoint5[18864] = {X 198.6105, Y 46.2305, Z -7.1667, A 0.000, B 0.000, C 0.000 }
gfCNCPoint5[18865] = {X 196.4933, Y 47.3403, Z -7.1667, A 0.000, B 0.000, C 0.000 }
gfCNCPoint5[18866] = {X 194.2898, Y 48.2674, Z -7.1667, A 0.000, B 0.000, C 0.000 }
gfCNCPoint5[18867] = {X 192.0159, Y 49.0049, Z -7.1667, A 0.000, B 0.000, C 0.000 }
gfCNCPoint5[18868] = {X 189.8185, Y 49.5138, Z -7.1667, A 0.000, B 0.000, C 0.000 }
gfCNCPoint5[18869] = {X 187.5807, Y 49.7977, Z -7.1667, A 0.000, B 0.000, C 0.000 }
gfCNCPoint5[18870] = {X 185.3258, Y 49.8536, Z -7.1667, A 0.000, B 0.000, C 0.000 }
gfCNCPoint5[18871] = {X 183.0768, Y 49.6808, Z -7.1667, A 0.000, B 0.000, C 0.000 }
gfCNCPoint5[18872] = {X 180.8568, Y 49.2813, Z -7.1667, A 0.000, B 0.000, C 0.000 }
gfCNCPoint5[18873] = {X 179.0341, Y 48.7530, Z -7.1667, A 0.000, B 0.000, C 0.000 }
gfCNCPoint5[18874] = {X 177.2845, Y 48.0181, Z -7.1667, A 0.000, B 0.000, C 0.000 }
gfCNCPoint5[18875] = {X 175.6313, Y 47.0863, Z -7.1667, A 0.000, B 0.000, C 0.000 }
gfCNCPoint5[18876] = {X 174.0965, Y 45.9701, Z -7.1667, A 0.000, B 0.000, C 0.000 }
gfCNCPoint5[18877] = {X 172.9699, Y 44.9422, Z -7.1667, A 0.000, B 0.000, C 0.000 }
gfCNCPoint5[18878] = {X 171.9728, Y 43.7883, Z -7.1667, A 0.000, B 0.000, C 0.000 }
gfCNCPoint5[18879] = {X 171.1192, Y 42.5244, Z -7.1667, A 0.000, B 0.000, C 0.000 }
gfCNCPoint5[18880] = {X 170.4212, Y 41.1685, Z -7.1667, A 0.000, B 0.000, C 0.000 }
gfCNCPoint5[18881] = {X 169.8885, Y 39.7394, Z -7.1667, A 0.000, B 0.000, C 0.000 }
gfCNCPoint5[18882] = {X 169.5286, Y 38.2574, Z -7.1667, A 0.000, B 0.000, C 0.000 }
gfCNCPoint5[18883] = {X 169.4733, Y 37.9104, Z -7.1667, A 0.000, B 0.000, C 0.000 }
gfCNCPoint5[18884] = {X 165.5231, Y 38.5394, Z -7.1667, A 0.000, B 0.000, C 0.000 }
gfCNCPoint5[18885] = {X 169.5523, Y 37.8978, Z -7.1667, A 0.000, B 0.000, C 0.000 }
gfCNCPoint5[18886] = {X 169.4970, Y 37.5504, Z -7.1667, A 0.000, B 0.000, C 0.000 }
gfCNCPoint5[18887] = {X 169.3415, Y 35.9716, Z -7.1667, A 0.000, B 0.000, C 0.000 }
gfCNCPoint5[18888] = {X 169.3584, Y 34.3853, Z -7.1667, A 0.000, B 0.000, C 0.000 }
gfCNCPoint5[18889] = {X 169.5475, Y 32.8101, Z -7.1667, A 0.000, B 0.000, C 0.000 }
gfCNCPoint5[18890] = {X 169.9067, Y 31.2649, Z -7.1667, A 0.000, B 0.000, C 0.000 }
gfCNCPoint5[18891] = {X 170.4315, Y 29.7677, Z -7.1667, A 0.000, B 0.000, C 0.000 }
gfCNCPoint5[18892] = {X 171.1145, Y 28.3891, Z -7.1667, A 0.000, B 0.000, C 0.000 }
gfCNCPoint5[18893] = {X 171.9896, Y 27.1237, Z -7.1667, A 0.000, B 0.000, C 0.000 }
gfCNCPoint5[18894] = {X 173.0385, Y 25.9981, Z -7.1667, A 0.000, B 0.000, C 0.000 }
gfCNCPoint5[18895] = {X 174.2391, Y 25.0360, Z -7.1667, A 0.000, B 0.000, C 0.000 }
gfCNCPoint5[18896] = {X 175.5662, Y 24.2576, Z -7.1667, A 0.000, B 0.000, C 0.000 }
gfCNCPoint5[18897] = {X 174.6543, Y 23.9377, Z -7.1667, A 0.000, B 0.000, C 0.000 }
gfCNCPoint5[18898] = {X 173.8433, Y 23.4124, Z -7.1667, A 0.000, B 0.000, C 0.000 }
gfCNCPoint5[18899] = {X 173.1785, Y 22.7111, Z -7.1667, A 0.000, B 0.000, C 0.000 }
gfCNCPoint5[18900] = {X 172.6973, Y 21.8731, Z -7.1667, A 0.000, B 0.000, C 0.000 }
gfCNCPoint5[18901] = {X 170.0626, Y 15.4213, Z -7.1667, A 0.000, B 0.000, C 0.000 }
gfCNCPoint5[18902] = {X 169.8043, Y 14.4793, Z -7.1667, A 0.000, B 0.000, C 0.000 }
gfCNCPoint5[18903] = {X 169.7773, Y 13.5028, Z -7.1667, A 0.000, B 0.000, C 0.000 }
gfCNCPoint5[18904] = {X 169.9832, Y 12.5479, Z -7.1667, A 0.000, B 0.000, C 0.000 }
gfCNCPoint5[18905] = {X 170.4102, Y 11.6694, Z -7.1667, A 0.000, B 0.000, C 0.000 }
gfCNCPoint5[18906] = {X 171.0337, Y 10.9174, Z -7.1667, A 0.000, B 0.000, C 0.000 }
gfCNCPoint5[18907] = {X 171.8181, Y 10.3353, Z -7.1667, A 0.000, B 0.000, C 0.000 }
gfCNCPoint5[18908] = {X 172.4475, Y 9.9764, Z -7.1667, A 0.000, B 0.000, C 0.000 }
gfCNCPoint5[18909] = {X 173.2688, Y 9.6293, Z -7.1667, A 0.000, B 0.000, C 0.000 }
gfCNCPoint5[18910] = {X 174.1459, Y 9.4689, Z -7.1667, A 0.000, B 0.000, C 0.000 }
gfCNCPoint5[18911] = {X 175.0368, Y 9.5028, Z -7.1667, A 0.000, B 0.000, C 0.000 }
gfCNCPoint5[18912] = {X 175.8992, Y 9.7295, Z -7.1667, A 0.000, B 0.000, C 0.000 }
gfCNCPoint5[18913] = {X 175.9646, Y 9.7552, Z -7.1667, A 0.000, B 0.000, C 0.000 }
gfCNCPoint5[18914] = {X 176.0296, Y 9.7821, Z -7.1667, A 0.000, B 0.000, C 0.000 }
gfCNCPoint5[18915] = {X 176.0573, Y 9.7600, Z -7.1667, A 0.000, B 0.000, C 0.000 }
gfCNCPoint5[18916] = {X 177.2217, Y 9.2648, Z -7.1667, A 0.000, B 0.000, C 0.000 }
gfCNCPoint5[18917] = {X 179.3694, Y 8.4743, Z -7.1667, A 0.000, B 0.000, C 0.000 }
gfCNCPoint5[18918] = {X 181.5845, Y 7.8995, Z -7.1667, A 0.000, B 0.000, C 0.000 }
gfCNCPoint5[18919] = {X 183.8456, Y 7.5461, Z -7.1667, A 0.000, B 0.000, C 0.000 }
gfCNCPoint5[18920] = {X 186.1305, Y 7.4175, Z -7.1667, A 0.000, B 0.000, C 0.000 }
gfCNCPoint5[18921] = {X 188.4169, Y 7.5150, Z -7.1667, A 0.000, B 0.000, C 0.000 }
gfCNCPoint5[18922] = {X 190.6825, Y 7.8376, Z -7.1667, A 0.000, B 0.000, C 0.000 }
gfCNCPoint5[18923] = {X 192.2491, Y 8.2187, Z -7.1667, A 0.000, B 0.000, C 0.000 }
gfCNCPoint5[18924] = {X 193.7721, Y 8.7477, Z -7.1667, A 0.000, B 0.000, C 0.000 }
gfCNCPoint5[18925] = {X 195.2375, Y 9.4199, Z -7.1667, A 0.000, B 0.000, C 0.000 }
gfCNCPoint5[18926] = {X 196.6321, Y 10.2289, Z -7.1667, A 0.000, B 0.000, C 0.000 }
gfCNCPoint5[18927] = {X 197.9430, Y 11.1675, Z -7.1667, A 0.000, B 0.000, C 0.000 }
gfCNCPoint5[18928] = {X 199.2267, Y 12.3413, Z -7.1667, A 0.000, B 0.000, C 0.000 }
gfCNCPoint5[18929] = {X 200.3391, Y 13.6786, Z -7.1667, A 0.000, B 0.000, C 0.000 }
gfCNCPoint5[18930] = {X 201.2597, Y 15.1545, Z -7.1667, A 0.000, B 0.000, C 0.000 }
gfCNCPoint5[18931] = {X 201.9714, Y 16.7417, Z -7.1667, A 0.000, B 0.000, C 0.000 }
gfCNCPoint5[18932] = {X 202.4376, Y 18.3713, Z -7.1667, A 0.000, B 0.000, C 0.000 }
gfCNCPoint5[18933] = {X 202.7143, Y 20.0435, Z -7.1667, A 0.000, B 0.000, C 0.000 }
gfCNCPoint5[18934] = {X 202.7977, Y 21.7363, Z -7.1667, A 0.000, B 0.000, C 0.000 }
gfCNCPoint5[18935] = {X 202.6868, Y 23.4277, Z -7.1667, A 0.000, B 0.000, C 0.000 }
gfCNCPoint5[18936] = {X 202.3830, Y 25.0951, Z -7.1667, A 0.000, B 0.000, C 0.000 }
gfCNCPoint5[18937] = {X 201.9158, Y 26.6018, Z -7.1667, A 0.000, B 0.000, C 0.000 }
gfCNCPoint5[18938] = {X 201.2460, Y 28.0301, Z -7.1667, A 0.000, B 0.000, C 0.000 }
gfCNCPoint5[18939] = {X 200.3863, Y 29.3527, Z -7.1667, A 0.000, B 0.000, C 0.000 }
gfCNCPoint5[18940] = {X 199.3531, Y 30.5448, Z -7.1667, A 0.000, B 0.000, C 0.000 }
gfCNCPoint5[18941] = {X 198.1660, Y 31.5836, Z -7.1667, A 0.000, B 0.000, C 0.000 }
gfCNCPoint5[18942] = {X 199.0636, Y 31.8624, Z -7.1667, A 0.000, B 0.000, C 0.000 }
gfCNCPoint5[18943] = {X 199.8736, Y 32.3393, Z -7.1667, A 0.000, B 0.000, C 0.000 }
gfCNCPoint5[18944] = {X 200.5530, Y 32.9888, Z -7.1667, A 0.000, B 0.000, C 0.000 }
gfCNCPoint5[18945] = {X 201.0657, Y 33.7766, Z -7.1667, A 0.000, B 0.000, C 0.000 }
gfCNCPoint5[18946] = {X 204.1061, Y 40.0576, Z -7.1667, A 0.000, B 0.000, C 0.000 }
gfCNCPoint5[18947] = {X 204.4089, Y 40.9162, Z -7.1667, A 0.000, B 0.000, C 0.000 }
gfCNCPoint5[18948] = {X 204.5137, Y 41.8206, Z -7.1667, A 0.000, B 0.000, C 0.000 }
gfCNCPoint5[18949] = {X 204.4154, Y 42.7257, Z -7.1667, A 0.000, B 0.000, C 0.000 }
gfCNCPoint5[18950] = {X 204.1188, Y 43.5864, Z -7.1667, A 0.000, B 0.000, C 0.000 }
gfCNCPoint5[18951] = {X 203.6387, Y 44.3600, Z -7.1667, A 0.000, B 0.000, C 0.000 }
gfCNCPoint5[18952] = {X 202.9990, Y 45.0078, Z -7.1667, A 0.000, B 0.000, C 0.000 }
gfCNCPoint5[18953] = {X 202.4628, Y 45.4413, Z -7.1667, A 0.000, B 0.000, C 0.000 }
gfCNCPoint5[18954] = {X 201.7791, Y 45.8891, Z -7.1667, A 0.000, B 0.000, C 0.000 }
gfCNCPoint5[18955] = {X 201.0201, Y 46.1921, Z -7.1667, A 0.000, B 0.000, C 0.000 }
gfCNCPoint5[18956] = {X 200.2160, Y 46.3383, Z -7.1667, A 0.000, B 0.000, C 0.000 }
gfCNCPoint5[18957] = {X 199.3989, Y 46.3218, Z -7.1667, A 0.000, B 0.000, C 0.000 }
gfCNCPoint5[18958] = {X 198.6013, Y 46.1433, Z -7.1667, A 0.000, B 0.000, C 0.000 }
gfCNCPoint5[18959] = {X 196.4806, Y 47.2578, Z -7.1667, A 0.000, B 0.000, C 0.000 }
gfCNCPoint5[18960] = {X 194.2729, Y 48.1883, Z -7.1667, A 0.000, B 0.000, C 0.000 }
gfCNCPoint5[18961] = {X 191.9942, Y 48.9279, Z -7.1667, A 0.000, B 0.000, C 0.000 }
gfCNCPoint5[18962] = {X 189.8046, Y 49.4351, Z -7.1667, A 0.000, B 0.000, C 0.000 }
gfCNCPoint5[18963] = {X 187.5748, Y 49.7179, Z -7.1667, A 0.000, B 0.000, C 0.000 }
gfCNCPoint5[18964] = {X 185.3279, Y 49.7736, Z -7.1667, A 0.000, B 0.000, C 0.000 }
gfCNCPoint5[18965] = {X 183.0869, Y 49.6015, Z -7.1667, A 0.000, B 0.000, C 0.000 }
gfCNCPoint5[18966] = {X 180.8748, Y 49.2033, Z -7.1667, A 0.000, B 0.000, C 0.000 }
gfCNCPoint5[18967] = {X 179.0609, Y 48.6776, Z -7.1667, A 0.000, B 0.000, C 0.000 }
gfCNCPoint5[18968] = {X 177.3197, Y 47.9462, Z -7.1667, A 0.000, B 0.000, C 0.000 }
gfCNCPoint5[18969] = {X 175.6744, Y 47.0189, Z -7.1667, A 0.000, B 0.000, C 0.000 }
gfCNCPoint5[18970] = {X 174.1471, Y 45.9081, Z -7.1667, A 0.000, B 0.000, C 0.000 }
gfCNCPoint5[18971] = {X 173.0275, Y 44.8867, Z -7.1667, A 0.000, B 0.000, C 0.000 }
gfCNCPoint5[18972] = {X 172.0366, Y 43.7400, Z -7.1667, A 0.000, B 0.000, C 0.000 }
gfCNCPoint5[18973] = {X 171.1883, Y 42.4841, Z -7.1667, A 0.000, B 0.000, C 0.000 }
gfCNCPoint5[18974] = {X 170.4946, Y 41.1367, Z -7.1667, A 0.000, B 0.000, C 0.000 }
gfCNCPoint5[18975] = {X 169.9652, Y 39.7167, Z -7.1667, A 0.000, B 0.000, C 0.000 }
gfCNCPoint5[18976] = {X 169.6074, Y 38.2440, Z -7.1667, A 0.000, B 0.000, C 0.000 }
gfCNCPoint5[18977] = {X 169.5523, Y 37.8978, Z -7.1667, A 0.000, B 0.000, C 0.000 }
gfCNCPoint5[18978] = {X 165.6021, Y 38.5268, Z -7.1667, A 0.000, B 0.000, C 0.000 }
gfCNCPoint5[18979] = {X 169.6313, Y 37.8853, Z -7.1667, A 0.000, B 0.000, C 0.000 }
gfCNCPoint5[18980] = {X 169.5761, Y 37.5383, Z -7.1667, A 0.000, B 0.000, C 0.000 }
gfCNCPoint5[18981] = {X 169.4214, Y 35.9681, Z -7.1667, A 0.000, B 0.000, C 0.000 }
gfCNCPoint5[18982] = {X 169.4383, Y 34.3904, Z -7.1667, A 0.000, B 0.000, C 0.000 }
gfCNCPoint5[18983] = {X 169.6264, Y 32.8239, Z -7.1667, A 0.000, B 0.000, C 0.000 }
gfCNCPoint5[18984] = {X 169.9835, Y 31.2871, Z -7.1667, A 0.000, B 0.000, C 0.000 }
gfCNCPoint5[18985] = {X 170.5055, Y 29.7981, Z -7.1667, A 0.000, B 0.000, C 0.000 }
gfCNCPoint5[18986] = {X 171.2080, Y 28.3881, Z -7.1667, A 0.000, B 0.000, C 0.000 }
gfCNCPoint5[18987] = {X 172.1130, Y 27.0987, Z -7.1667, A 0.000, B 0.000, C 0.000 }
gfCNCPoint5[18988] = {X 173.2002, Y 25.9586, Z -7.1667, A 0.000, B 0.000, C 0.000 }
gfCNCPoint5[18989] = {X 174.4452, Y 24.9934, Z -7.1667, A 0.000, B 0.000, C 0.000 }
gfCNCPoint5[18990] = {X 175.8202, Y 24.2246, Z -7.1667, A 0.000, B 0.000, C 0.000 }
gfCNCPoint5[18991] = {X 175.0295, Y 24.0136, Z -7.1667, A 0.000, B 0.000, C 0.000 }
gfCNCPoint5[18992] = {X 174.2983, Y 23.6460, Z -7.1667, A 0.000, B 0.000, C 0.000 }
gfCNCPoint5[18993] = {X 173.6573, Y 23.1372, Z -7.1667, A 0.000, B 0.000, C 0.000 }
gfCNCPoint5[18994] = {X 173.1332, Y 22.5087, Z -7.1667, A 0.000, B 0.000, C 0.000 }
gfCNCPoint5[18995] = {X 172.7479, Y 21.7866, Z -7.1667, A 0.000, B 0.000, C 0.000 }
gfCNCPoint5[18996] = {X 170.1367, Y 15.3911, Z -7.1667, A 0.000, B 0.000, C 0.000 }
gfCNCPoint5[18997] = {X 169.8835, Y 14.4675, Z -7.1667, A 0.000, B 0.000, C 0.000 }
gfCNCPoint5[18998] = {X 169.8570, Y 13.5102, Z -7.1667, A 0.000, B 0.000, C 0.000 }
gfCNCPoint5[18999] = {X 170.0588, Y 12.5740, Z -7.1667, A 0.000, B 0.000, C 0.000 }
gfCNCPoint5[19000] = {X 170.4774, Y 11.7127, Z -7.1667, A 0.000, B 0.000, C 0.000 }
gfCNCPoint5[19001] = {X 171.0888, Y 10.9755, Z -7.1667, A 0.000, B 0.000, C 0.000 }
gfCNCPoint5[19002] = {X 171.8578, Y 10.4048, Z -7.1667, A 0.000, B 0.000, C 0.000 }
gfCNCPoint5[19003] = {X 172.4867, Y 10.0462, Z -7.1667, A 0.000, B 0.000, C 0.000 }
gfCNCPoint5[19004] = {X 173.2918, Y 9.7059, Z -7.1667, A 0.000, B 0.000, C 0.000 }
gfCNCPoint5[19005] = {X 174.1517, Y 9.5487, Z -7.1667, A 0.000, B 0.000, C 0.000 }
gfCNCPoint5[19006] = {X 175.0251, Y 9.5819, Z -7.1667, A 0.000, B 0.000, C 0.000 }
gfCNCPoint5[19007] = {X 175.8705, Y 9.8041, Z -7.1667, A 0.000, B 0.000, C 0.000 }
gfCNCPoint5[19008] = {X 175.9567, Y 9.8384, Z -7.1667, A 0.000, B 0.000, C 0.000 }
gfCNCPoint5[19009] = {X 176.0421, Y 9.8746, Z -7.1667, A 0.000, B 0.000, C 0.000 }
gfCNCPoint5[19010] = {X 176.0987, Y 9.8293, Z -7.1667, A 0.000, B 0.000, C 0.000 }
gfCNCPoint5[19011] = {X 177.2531, Y 9.3384, Z -7.1667, A 0.000, B 0.000, C 0.000 }
gfCNCPoint5[19012] = {X 179.3933, Y 8.5506, Z -7.1667, A 0.000, B 0.000, C 0.000 }
gfCNCPoint5[19013] = {X 181.6008, Y 7.9779, Z -7.1667, A 0.000, B 0.000, C 0.000 }
gfCNCPoint5[19014] = {X 183.8540, Y 7.6257, Z -7.1667, A 0.000, B 0.000, C 0.000 }
gfCNCPoint5[19015] = {X 186.1310, Y 7.4975, Z -7.1667, A 0.000, B 0.000, C 0.000 }
gfCNCPoint5[19016] = {X 188.4095, Y 7.5947, Z -7.1667, A 0.000, B 0.000, C 0.000 }
gfCNCPoint5[19017] = {X 190.6674, Y 7.9161, Z -7.1667, A 0.000, B 0.000, C 0.000 }
gfCNCPoint5[19018] = {X 192.6100, Y 8.4134, Z -7.1667, A 0.000, B 0.000, C 0.000 }
gfCNCPoint5[19019] = {X 194.4795, Y 9.1390, Z -7.1667, A 0.000, B 0.000, C 0.000 }
gfCNCPoint5[19020] = {X 196.2490, Y 10.0824, Z -7.1667, A 0.000, B 0.000, C 0.000 }
gfCNCPoint5[19021] = {X 197.8934, Y 11.2302, Z -7.1667, A 0.000, B 0.000, C 0.000 }
gfCNCPoint5[19022] = {X 199.1688, Y 12.3966, Z -7.1667, A 0.000, B 0.000, C 0.000 }
gfCNCPoint5[19023] = {X 200.2741, Y 13.7253, Z -7.1667, A 0.000, B 0.000, C 0.000 }
gfCNCPoint5[19024] = {X 201.1889, Y 15.1917, Z -7.1667, A 0.000, B 0.000, C 0.000 }
gfCNCPoint5[19025] = {X 201.8961, Y 16.7687, Z -7.1667, A 0.000, B 0.000, C 0.000 }
gfCNCPoint5[19026] = {X 202.3597, Y 18.3894, Z -7.1667, A 0.000, B 0.000, C 0.000 }
gfCNCPoint5[19027] = {X 202.6348, Y 20.0525, Z -7.1667, A 0.000, B 0.000, C 0.000 }
gfCNCPoint5[19028] = {X 202.7177, Y 21.7361, Z -7.1667, A 0.000, B 0.000, C 0.000 }
gfCNCPoint5[19029] = {X 202.6074, Y 23.4182, Z -7.1667, A 0.000, B 0.000, C 0.000 }
gfCNCPoint5[19030] = {X 202.3052, Y 25.0766, Z -7.1667, A 0.000, B 0.000, C 0.000 }
gfCNCPoint5[19031] = {X 201.8277, Y 26.6077, Z -7.1667, A 0.000, B 0.000, C 0.000 }
gfCNCPoint5[19032] = {X 201.1395, Y 28.0565, Z -7.1667, A 0.000, B 0.000, C 0.000 }
gfCNCPoint5[19033] = {X 200.2544, Y 29.3941, Z -7.1667, A 0.000, B 0.000, C 0.000 }
gfCNCPoint5[19034] = {X 199.1900, Y 30.5939, Z -7.1667, A 0.000, B 0.000, C 0.000 }
gfCNCPoint5[19035] = {X 197.9674, Y 31.6321, Z -7.1667, A 0.000, B 0.000, C 0.000 }
gfCNCPoint5[19036] = {X 198.7289, Y 31.8162, Z -7.1667, A 0.000, B 0.000, C 0.000 }
gfCNCPoint5[19037] = {X 199.4398, Y 32.1452, Z -7.1667, A 0.000, B 0.000, C 0.000 }
gfCNCPoint5[19038] = {X 200.0730, Y 32.6065, Z -7.1667, A 0.000, B 0.000, C 0.000 }
gfCNCPoint5[19039] = {X 200.6042, Y 33.1824, Z -7.1667, A 0.000, B 0.000, C 0.000 }
gfCNCPoint5[19040] = {X 201.0129, Y 33.8507, Z -7.1667, A 0.000, B 0.000, C 0.000 }
gfCNCPoint5[19041] = {X 204.0341, Y 40.0925, Z -7.1667, A 0.000, B 0.000, C 0.000 }
gfCNCPoint5[19042] = {X 204.3309, Y 40.9342, Z -7.1667, A 0.000, B 0.000, C 0.000 }
gfCNCPoint5[19043] = {X 204.4337, Y 41.8209, Z -7.1667, A 0.000, B 0.000, C 0.000 }
gfCNCPoint5[19044] = {X 204.3373, Y 42.7082, Z -7.1667, A 0.000, B 0.000, C 0.000 }
gfCNCPoint5[19045] = {X 204.0465, Y 43.5521, Z -7.1667, A 0.000, B 0.000, C 0.000 }
gfCNCPoint5[19046] = {X 203.5758, Y 44.3105, Z -7.1667, A 0.000, B 0.000, C 0.000 }
gfCNCPoint5[19047] = {X 202.9487, Y 44.9456, Z -7.1667, A 0.000, B 0.000, C 0.000 }
gfCNCPoint5[19048] = {X 202.4125, Y 45.3791, Z -7.1667, A 0.000, B 0.000, C 0.000 }
gfCNCPoint5[19049] = {X 201.7358, Y 45.8215, Z -7.1667, A 0.000, B 0.000, C 0.000 }
gfCNCPoint5[19050] = {X 200.9842, Y 46.1192, Z -7.1667, A 0.000, B 0.000, C 0.000 }
gfCNCPoint5[19051] = {X 200.1881, Y 46.2602, Z -7.1667, A 0.000, B 0.000, C 0.000 }
gfCNCPoint5[19052] = {X 199.3800, Y 46.2388, Z -7.1667, A 0.000, B 0.000, C 0.000 }
gfCNCPoint5[19053] = {X 198.5925, Y 46.0559, Z -7.1667, A 0.000, B 0.000, C 0.000 }
gfCNCPoint5[19054] = {X 196.4682, Y 47.1752, Z -7.1667, A 0.000, B 0.000, C 0.000 }
gfCNCPoint5[19055] = {X 194.2562, Y 48.1092, Z -7.1667, A 0.000, B 0.000, C 0.000 }
gfCNCPoint5[19056] = {X 191.9725, Y 48.8509, Z -7.1667, A 0.000, B 0.000, C 0.000 }
gfCNCPoint5[19057] = {X 189.7907, Y 49.3563, Z -7.1667, A 0.000, B 0.000, C 0.000 }
gfCNCPoint5[19058] = {X 187.5689, Y 49.6381, Z -7.1667, A 0.000, B 0.000, C 0.000 }
gfCNCPoint5[19059] = {X 185.3300, Y 49.6936, Z -7.1667, A 0.000, B 0.000, C 0.000 }
gfCNCPoint5[19060] = {X 183.0969, Y 49.5221, Z -7.1667, A 0.000, B 0.000, C 0.000 }
gfCNCPoint5[19061] = {X 180.8928, Y 49.1254, Z -7.1667, A 0.000, B 0.000, C 0.000 }
gfCNCPoint5[19062] = {X 179.0876, Y 48.6022, Z -7.1667, A 0.000, B 0.000, C 0.000 }
gfCNCPoint5[19063] = {X 177.3548, Y 47.8744, Z -7.1667, A 0.000, B 0.000, C 0.000 }
gfCNCPoint5[19064] = {X 175.7175, Y 46.9515, Z -7.1667, A 0.000, B 0.000, C 0.000 }
gfCNCPoint5[19065] = {X 174.1976, Y 45.8461, Z -7.1667, A 0.000, B 0.000, C 0.000 }
gfCNCPoint5[19066] = {X 173.0851, Y 44.8312, Z -7.1667, A 0.000, B 0.000, C 0.000 }
gfCNCPoint5[19067] = {X 172.1004, Y 43.6917, Z -7.1667, A 0.000, B 0.000, C 0.000 }
gfCNCPoint5[19068] = {X 171.2574, Y 42.4438, Z -7.1667, A 0.000, B 0.000, C 0.000 }
gfCNCPoint5[19069] = {X 170.5680, Y 41.1050, Z -7.1667, A 0.000, B 0.000, C 0.000 }
gfCNCPoint5[19070] = {X 170.0419, Y 39.6940, Z -7.1667, A 0.000, B 0.000, C 0.000 }
gfCNCPoint5[19071] = {X 169.6863, Y 38.2306, Z -7.1667, A 0.000, B 0.000, C 0.000 }
gfCNCPoint5[19072] = {X 169.6313, Y 37.8853, Z -7.1667, A 0.000, B 0.000, C 0.000 }
gfCNCPoint5[19073] = {X 165.6021, Y 38.5268, Z -7.1667, A 0.000, B 0.000, C 0.000 }
gfCNCPoint5[19074] = {X 165.6021, Y 38.5268, Z -4.1667, A 0.000, B 0.000, C 0.000 }
gfCNCPoint5[19075] = {X 165.6021, Y 38.5268, Z 11.0000, A 0.000, B 0.000, C 0.000 }
gfCNCPoint5[19076] = {X 210.1639, Y 28.5737, Z 11.0000, A 0.000, B 0.000, C 0.000 }
gfCNCPoint5[19077] = {X 210.1639, Y 28.5737, Z -4.1667, A 0.000, B 0.000, C 0.000 }
gfCNCPoint5[19078] = {X 210.1639, Y 28.5737, Z -7.1667, A 0.000, B 0.000, C 0.000 }
gfCNCPoint5[19079] = {X 214.2439, Y 28.5737, Z -7.1667, A 0.000, B 0.000, C 0.000 }
gfCNCPoint5[19080] = {X 214.2439, Y 17.4624, Z -7.1667, A 0.000, B 0.000, C 0.000 }
gfCNCPoint5[19081] = {X 214.2385, Y 16.7692, Z -7.1667, A 0.000, B 0.000, C 0.000 }
gfCNCPoint5[19082] = {X 214.2420, Y 16.2720, Z -7.1667, A 0.000, B 0.000, C 0.000 }
gfCNCPoint5[19083] = {X 213.6044, Y 15.6009, Z -7.1667, A 0.000, B 0.000, C 0.000 }
gfCNCPoint5[19084] = {X 213.1244, Y 14.8093, Z -7.1667, A 0.000, B 0.000, C 0.000 }
gfCNCPoint5[19085] = {X 212.8240, Y 13.9337, Z -7.1667, A 0.000, B 0.000, C 0.000 }
gfCNCPoint5[19086] = {X 212.7172, Y 13.0141, Z -7.1667, A 0.000, B 0.000, C 0.000 }
gfCNCPoint5[19087] = {X 212.7170, Y 12.1868, Z -7.1667, A 0.000, B 0.000, C 0.000 }
gfCNCPoint5[19088] = {X 212.8253, Y 11.2255, Z -7.1667, A 0.000, B 0.000, C 0.000 }
gfCNCPoint5[19089] = {X 213.1448, Y 10.3124, Z -7.1667, A 0.000, B 0.000, C 0.000 }
gfCNCPoint5[19090] = {X 213.6595, Y 9.4933, Z -7.1667, A 0.000, B 0.000, C 0.000 }
gfCNCPoint5[19091] = {X 214.3435, Y 8.8093, Z -7.1667, A 0.000, B 0.000, C 0.000 }
gfCNCPoint5[19092] = {X 215.1626, Y 8.2946, Z -7.1667, A 0.000, B 0.000, C 0.000 }
gfCNCPoint5[19093] = {X 216.0757, Y 7.9751, Z -7.1667, A 0.000, B 0.000, C 0.000 }
gfCNCPoint5[19094] = {X 217.0370, Y 7.8668, Z -7.1667, A 0.000, B 0.000, C 0.000 }
gfCNCPoint5[19095] = {X 223.4805, Y 7.8668, Z -7.1667, A 0.000, B 0.000, C 0.000 }
gfCNCPoint5[19096] = {X 224.4418, Y 7.9751, Z -7.1667, A 0.000, B 0.000, C 0.000 }
gfCNCPoint5[19097] = {X 225.3549, Y 8.2946, Z -7.1667, A 0.000, B 0.000, C 0.000 }
gfCNCPoint5[19098] = {X 226.1740, Y 8.8093, Z -7.1667, A 0.000, B 0.000, C 0.000 }
gfCNCPoint5[19099] = {X 226.8580, Y 9.4933, Z -7.1667, A 0.000, B 0.000, C 0.000 }
gfCNCPoint5[19100] = {X 227.3727, Y 10.3124, Z -7.1667, A 0.000, B 0.000, C 0.000 }
gfCNCPoint5[19101] = {X 227.6922, Y 11.2255, Z -7.1667, A 0.000, B 0.000, C 0.000 }
gfCNCPoint5[19102] = {X 227.8005, Y 12.1868, Z -7.1667, A 0.000, B 0.000, C 0.000 }
gfCNCPoint5[19103] = {X 227.8005, Y 12.9782, Z -7.1667, A 0.000, B 0.000, C 0.000 }
gfCNCPoint5[19104] = {X 227.6992, Y 13.9078, Z -7.1667, A 0.000, B 0.000, C 0.000 }
gfCNCPoint5[19105] = {X 227.4003, Y 14.7938, Z -7.1667, A 0.000, B 0.000, C 0.000 }
gfCNCPoint5[19106] = {X 226.9178, Y 15.5948, Z -7.1667, A 0.000, B 0.000, C 0.000 }
gfCNCPoint5[19107] = {X 226.2741, Y 16.2731, Z -7.1667, A 0.000, B 0.000, C 0.000 }
gfCNCPoint5[19108] = {X 226.2751, Y 40.9156, Z -7.1667, A 0.000, B 0.000, C 0.000 }
gfCNCPoint5[19109] = {X 226.9121, Y 41.5858, Z -7.1667, A 0.000, B 0.000, C 0.000 }
gfCNCPoint5[19110] = {X 227.3920, Y 42.3762, Z -7.1667, A 0.000, B 0.000, C 0.000 }
gfCNCPoint5[19111] = {X 227.6926, Y 43.2506, Z -7.1667, A 0.000, B 0.000, C 0.000 }
gfCNCPoint5[19112] = {X 227.8003, Y 44.1689, Z -7.1667, A 0.000, B 0.000, C 0.000 }
gfCNCPoint5[19113] = {X 227.8005, Y 45.0000, Z -7.1667, A 0.000, B 0.000, C 0.000 }
gfCNCPoint5[19114] = {X 227.6922, Y 45.9613, Z -7.1667, A 0.000, B 0.000, C 0.000 }
gfCNCPoint5[19115] = {X 227.3727, Y 46.8744, Z -7.1667, A 0.000, B 0.000, C 0.000 }
gfCNCPoint5[19116] = {X 226.8580, Y 47.6935, Z -7.1667, A 0.000, B 0.000, C 0.000 }
gfCNCPoint5[19117] = {X 226.1740, Y 48.3775, Z -7.1667, A 0.000, B 0.000, C 0.000 }
gfCNCPoint5[19118] = {X 225.3549, Y 48.8922, Z -7.1667, A 0.000, B 0.000, C 0.000 }
gfCNCPoint5[19119] = {X 224.4418, Y 49.2117, Z -7.1667, A 0.000, B 0.000, C 0.000 }
gfCNCPoint5[19120] = {X 223.4805, Y 49.3200, Z -7.1667, A 0.000, B 0.000, C 0.000 }
gfCNCPoint5[19121] = {X 217.0370, Y 49.3200, Z -7.1667, A 0.000, B 0.000, C 0.000 }
gfCNCPoint5[19122] = {X 216.0805, Y 49.2128, Z -7.1667, A 0.000, B 0.000, C 0.000 }
gfCNCPoint5[19123] = {X 215.1715, Y 48.8964, Z -7.1667, A 0.000, B 0.000, C 0.000 }
gfCNCPoint5[19124] = {X 214.3551, Y 48.3867, Z -7.1667, A 0.000, B 0.000, C 0.000 }
gfCNCPoint5[19125] = {X 213.6718, Y 47.7088, Z -7.1667, A 0.000, B 0.000, C 0.000 }
gfCNCPoint5[19126] = {X 213.1556, Y 46.8965, Z -7.1667, A 0.000, B 0.000, C 0.000 }
gfCNCPoint5[19127] = {X 212.8320, Y 45.9901, Z -7.1667, A 0.000, B 0.000, C 0.000 }
gfCNCPoint5[19128] = {X 212.7172, Y 45.0345, Z -7.1667, A 0.000, B 0.000, C 0.000 }
gfCNCPoint5[19129] = {X 212.7170, Y 44.1909, Z -7.1667, A 0.000, B 0.000, C 0.000 }
gfCNCPoint5[19130] = {X 212.7887, Y 43.4145, Z -7.1667, A 0.000, B 0.000, C 0.000 }
gfCNCPoint5[19131] = {X 213.0013, Y 42.6644, Z -7.1667, A 0.000, B 0.000, C 0.000 }
gfCNCPoint5[19132] = {X 213.3476, Y 41.9658, Z -7.1667, A 0.000, B 0.000, C 0.000 }
gfCNCPoint5[19133] = {X 213.8160, Y 41.3425, Z -7.1667, A 0.000, B 0.000, C 0.000 }
gfCNCPoint5[19134] = {X 214.2395, Y 40.8754, Z -7.1667, A 0.000, B 0.000, C 0.000 }
gfCNCPoint5[19135] = {X 214.2439, Y 40.3062, Z -7.1667, A 0.000, B 0.000, C 0.000 }
gfCNCPoint5[19136] = {X 214.2439, Y 28.5737, Z -7.1667, A 0.000, B 0.000, C 0.000 }
gfCNCPoint5[19137] = {X 210.2439, Y 28.5737, Z -7.1667, A 0.000, B 0.000, C 0.000 }
gfCNCPoint5[19138] = {X 214.3239, Y 28.5737, Z -7.1667, A 0.000, B 0.000, C 0.000 }
gfCNCPoint5[19139] = {X 214.3239, Y 17.4621, Z -7.1667, A 0.000, B 0.000, C 0.000 }
gfCNCPoint5[19140] = {X 214.3185, Y 16.7691, Z -7.1667, A 0.000, B 0.000, C 0.000 }
gfCNCPoint5[19141] = {X 214.3223, Y 16.2350, Z -7.1667, A 0.000, B 0.000, C 0.000 }
gfCNCPoint5[19142] = {X 213.6850, Y 15.5745, Z -7.1667, A 0.000, B 0.000, C 0.000 }
gfCNCPoint5[19143] = {X 213.2048, Y 14.7923, Z -7.1667, A 0.000, B 0.000, C 0.000 }
gfCNCPoint5[19144] = {X 212.9041, Y 13.9251, Z -7.1667, A 0.000, B 0.000, C 0.000 }
gfCNCPoint5[19145] = {X 212.7972, Y 13.0135, Z -7.1667, A 0.000, B 0.000, C 0.000 }
gfCNCPoint5[19146] = {X 212.7970, Y 12.1868, Z -7.1667, A 0.000, B 0.000, C 0.000 }
gfCNCPoint5[19147] = {X 212.9033, Y 11.2433, Z -7.1667, A 0.000, B 0.000, C 0.000 }
gfCNCPoint5[19148] = {X 213.2169, Y 10.3472, Z -7.1667, A 0.000, B 0.000, C 0.000 }
gfCNCPoint5[19149] = {X 213.7220, Y 9.5432, Z -7.1667, A 0.000, B 0.000, C 0.000 }
gfCNCPoint5[19150] = {X 214.3934, Y 8.8719, Z -7.1667, A 0.000, B 0.000, C 0.000 }
gfCNCPoint5[19151] = {X 215.1973, Y 8.3667, Z -7.1667, A 0.000, B 0.000, C 0.000 }
gfCNCPoint5[19152] = {X 216.0935, Y 8.0531, Z -7.1667, A 0.000, B 0.000, C 0.000 }
gfCNCPoint5[19153] = {X 217.0370, Y 7.9468, Z -7.1667, A 0.000, B 0.000, C 0.000 }
gfCNCPoint5[19154] = {X 223.4805, Y 7.9468, Z -7.1667, A 0.000, B 0.000, C 0.000 }
gfCNCPoint5[19155] = {X 224.4240, Y 8.0531, Z -7.1667, A 0.000, B 0.000, C 0.000 }
gfCNCPoint5[19156] = {X 225.3201, Y 8.3667, Z -7.1667, A 0.000, B 0.000, C 0.000 }
gfCNCPoint5[19157] = {X 226.1241, Y 8.8718, Z -7.1667, A 0.000, B 0.000, C 0.000 }
gfCNCPoint5[19158] = {X 226.7954, Y 9.5432, Z -7.1667, A 0.000, B 0.000, C 0.000 }
gfCNCPoint5[19159] = {X 227.3006, Y 10.3471, Z -7.1667, A 0.000, B 0.000, C 0.000 }
gfCNCPoint5[19160] = {X 227.6142, Y 11.2433, Z -7.1667, A 0.000, B 0.000, C 0.000 }
gfCNCPoint5[19161] = {X 227.7205, Y 12.1868, Z -7.1667, A 0.000, B 0.000, C 0.000 }
gfCNCPoint5[19162] = {X 227.7205, Y 12.9782, Z -7.1667, A 0.000, B 0.000, C 0.000 }
gfCNCPoint5[19163] = {X 227.6191, Y 13.8996, Z -7.1667, A 0.000, B 0.000, C 0.000 }
gfCNCPoint5[19164] = {X 227.3199, Y 14.7769, Z -7.1667, A 0.000, B 0.000, C 0.000 }
gfCNCPoint5[19165] = {X 226.8373, Y 15.5683, Z -7.1667, A 0.000, B 0.000, C 0.000 }
gfCNCPoint5[19166] = {X 226.1941, Y 16.2359, Z -7.1667, A 0.000, B 0.000, C 0.000 }
gfCNCPoint5[19167] = {X 226.1951, Y 40.9529, Z -7.1667, A 0.000, B 0.000, C 0.000 }
gfCNCPoint5[19168] = {X 226.8317, Y 41.6124, Z -7.1667, A 0.000, B 0.000, C 0.000 }
gfCNCPoint5[19169] = {X 227.3117, Y 42.3934, Z -7.1667, A 0.000, B 0.000, C 0.000 }
gfCNCPoint5[19170] = {X 227.6126, Y 43.2593, Z -7.1667, A 0.000, B 0.000, C 0.000 }
gfCNCPoint5[19171] = {X 227.7203, Y 44.1697, Z -7.1667, A 0.000, B 0.000, C 0.000 }
gfCNCPoint5[19172] = {X 227.7205, Y 45.0000, Z -7.1667, A 0.000, B 0.000, C 0.000 }
gfCNCPoint5[19173] = {X 227.6142, Y 45.9435, Z -7.1667, A 0.000, B 0.000, C 0.000 }
gfCNCPoint5[19174] = {X 227.3006, Y 46.8397, Z -7.1667, A 0.000, B 0.000, C 0.000 }
gfCNCPoint5[19175] = {X 226.7954, Y 47.6436, Z -7.1667, A 0.000, B 0.000, C 0.000 }
gfCNCPoint5[19176] = {X 226.1241, Y 48.3150, Z -7.1667, A 0.000, B 0.000, C 0.000 }
gfCNCPoint5[19177] = {X 225.3201, Y 48.8201, Z -7.1667, A 0.000, B 0.000, C 0.000 }
gfCNCPoint5[19178] = {X 224.4240, Y 49.1337, Z -7.1667, A 0.000, B 0.000, C 0.000 }
gfCNCPoint5[19179] = {X 223.4805, Y 49.2400, Z -7.1667, A 0.000, B 0.000, C 0.000 }
gfCNCPoint5[19180] = {X 217.0370, Y 49.2400, Z -7.1667, A 0.000, B 0.000, C 0.000 }
gfCNCPoint5[19181] = {X 216.0982, Y 49.1348, Z -7.1667, A 0.000, B 0.000, C 0.000 }
gfCNCPoint5[19182] = {X 215.2061, Y 48.8243, Z -7.1667, A 0.000, B 0.000, C 0.000 }
gfCNCPoint5[19183] = {X 214.4048, Y 48.3240, Z -7.1667, A 0.000, B 0.000, C 0.000 }
gfCNCPoint5[19184] = {X 213.7341, Y 47.6587, Z -7.1667, A 0.000, B 0.000, C 0.000 }
gfCNCPoint5[19185] = {X 213.2275, Y 46.8614, Z -7.1667, A 0.000, B 0.000, C 0.000 }
gfCNCPoint5[19186] = {X 212.9099, Y 45.9717, Z -7.1667, A 0.000, B 0.000, C 0.000 }
gfCNCPoint5[19187] = {X 212.7972, Y 45.0338, Z -7.1667, A 0.000, B 0.000, C 0.000 }
gfCNCPoint5[19188] = {X 212.7970, Y 44.1909, Z -7.1667, A 0.000, B 0.000, C 0.000 }
gfCNCPoint5[19189] = {X 212.8673, Y 43.4292, Z -7.1667, A 0.000, B 0.000, C 0.000 }
gfCNCPoint5[19190] = {X 213.0759, Y 42.6932, Z -7.1667, A 0.000, B 0.000, C 0.000 }
gfCNCPoint5[19191] = {X 213.4157, Y 42.0078, Z -7.1667, A 0.000, B 0.000, C 0.000 }
gfCNCPoint5[19192] = {X 213.8753, Y 41.3962, Z -7.1667, A 0.000, B 0.000, C 0.000 }
gfCNCPoint5[19193] = {X 214.3193, Y 40.9065, Z -7.1667, A 0.000, B 0.000, C 0.000 }
gfCNCPoint5[19194] = {X 214.3239, Y 40.3065, Z -7.1667, A 0.000, B 0.000, C 0.000 }
gfCNCPoint5[19195] = {X 214.3239, Y 28.5737, Z -7.1667, A 0.000, B 0.000, C 0.000 }
gfCNCPoint5[19196] = {X 210.3239, Y 28.5737, Z -7.1667, A 0.000, B 0.000, C 0.000 }
gfCNCPoint5[19197] = {X 214.4039, Y 28.5737, Z -7.1667, A 0.000, B 0.000, C 0.000 }
gfCNCPoint5[19198] = {X 214.4039, Y 17.4617, Z -7.1667, A 0.000, B 0.000, C 0.000 }
gfCNCPoint5[19199] = {X 214.3985, Y 16.7691, Z -7.1667, A 0.000, B 0.000, C 0.000 }
gfCNCPoint5[19200] = {X 214.4025, Y 16.1975, Z -7.1667, A 0.000, B 0.000, C 0.000 }
gfCNCPoint5[19201] = {X 213.7656, Y 15.5477, Z -7.1667, A 0.000, B 0.000, C 0.000 }
gfCNCPoint5[19202] = {X 213.2852, Y 14.7750, Z -7.1667, A 0.000, B 0.000, C 0.000 }
gfCNCPoint5[19203] = {X 212.9842, Y 13.9164, Z -7.1667, A 0.000, B 0.000, C 0.000 }
gfCNCPoint5[19204] = {X 212.8772, Y 13.0128, Z -7.1667, A 0.000, B 0.000, C 0.000 }
gfCNCPoint5[19205] = {X 212.8770, Y 12.1868, Z -7.1667, A 0.000, B 0.000, C 0.000 }
gfCNCPoint5[19206] = {X 212.9813, Y 11.2611, Z -7.1667, A 0.000, B 0.000, C 0.000 }
gfCNCPoint5[19207] = {X 213.2890, Y 10.3819, Z -7.1667, A 0.000, B 0.000, C 0.000 }
gfCNCPoint5[19208] = {X 213.7846, Y 9.5931, Z -7.1667, A 0.000, B 0.000, C 0.000 }
gfCNCPoint5[19209] = {X 214.4433, Y 8.9344, Z -7.1667, A 0.000, B 0.000, C 0.000 }
gfCNCPoint5[19210] = {X 215.2321, Y 8.4388, Z -7.1667, A 0.000, B 0.000, C 0.000 }
gfCNCPoint5[19211] = {X 216.1113, Y 8.1311, Z -7.1667, A 0.000, B 0.000, C 0.000 }
gfCNCPoint5[19212] = {X 217.0370, Y 8.0268, Z -7.1667, A 0.000, B 0.000, C 0.000 }
gfCNCPoint5[19213] = {X 223.4805, Y 8.0268, Z -7.1667, A 0.000, B 0.000, C 0.000 }
gfCNCPoint5[19214] = {X 224.4062, Y 8.1311, Z -7.1667, A 0.000, B 0.000, C 0.000 }
gfCNCPoint5[19215] = {X 225.2854, Y 8.4388, Z -7.1667, A 0.000, B 0.000, C 0.000 }
gfCNCPoint5[19216] = {X 226.0742, Y 8.9344, Z -7.1667, A 0.000, B 0.000, C 0.000 }
gfCNCPoint5[19217] = {X 226.7329, Y 9.5931, Z -7.1667, A 0.000, B 0.000, C 0.000 }
gfCNCPoint5[19218] = {X 227.2285, Y 10.3819, Z -7.1667, A 0.000, B 0.000, C 0.000 }
gfCNCPoint5[19219] = {X 227.5362, Y 11.2611, Z -7.1667, A 0.000, B 0.000, C 0.000 }
gfCNCPoint5[19220] = {X 227.6405, Y 12.1868, Z -7.1667, A 0.000, B 0.000, C 0.000 }
gfCNCPoint5[19221] = {X 227.6405, Y 12.9782, Z -7.1667, A 0.000, B 0.000, C 0.000 }
gfCNCPoint5[19222] = {X 227.5390, Y 13.8913, Z -7.1667, A 0.000, B 0.000, C 0.000 }
gfCNCPoint5[19223] = {X 227.2395, Y 14.7599, Z -7.1667, A 0.000, B 0.000, C 0.000 }
gfCNCPoint5[19224] = {X 226.7567, Y 15.5416, Z -7.1667, A 0.000, B 0.000, C 0.000 }
gfCNCPoint5[19225] = {X 226.1141, Y 16.1982, Z -7.1667, A 0.000, B 0.000, C 0.000 }
gfCNCPoint5[19226] = {X 226.1151, Y 40.9906, Z -7.1667, A 0.000, B 0.000, C 0.000 }
gfCNCPoint5[19227] = {X 226.7512, Y 41.6394, Z -7.1667, A 0.000, B 0.000, C 0.000 }
gfCNCPoint5[19228] = {X 227.2313, Y 42.4109, Z -7.1667, A 0.000, B 0.000, C 0.000 }
gfCNCPoint5[19229] = {X 227.5325, Y 43.2682, Z -7.1667, A 0.000, B 0.000, C 0.000 }
gfCNCPoint5[19230] = {X 227.6403, Y 44.1704, Z -7.1667, A 0.000, B 0.000, C 0.000 }
